// TIA Portal V18 export
DATA_BLOCK "DB_ALL_PROCESS_PARAMETERS"   // DB5000
{ S7_Optimized_Access := 'TRUE' }
// stored: AutoNumber false, MemoryReserve 1000
   VAR RETAIN
      "Choosen Recipe Number" : Bool;
      ACTUAL_CHOOSEN_TYPE : "UDT_OP10_Recipe_type";   // THERE IS ASCTUAL DATA READED OUT FROM LIBRARY OF 20 TYPES BELOW
      PRODUCT_TYPE : Array[1..10] of "UDT_OP10_Recipe_type";   // PACK OF TWENTY DIFFERENT TYPES PRODUCT AND THEIR PARAMETERS FOR THE PROCESS
   END_VAR
BEGIN
   ACTUAL_CHOOSEN_TYPE.Header.RecipeName := 'produkt 1';
   ACTUAL_CHOOSEN_TYPE.Header.RecipeID := 2;
   ACTUAL_CHOOSEN_TYPE.Header."Version" := 19629;
   ACTUAL_CHOOSEN_TYPE.Header.LastModified := DTL#2026-01-17-04:23:27.501;
   ACTUAL_CHOOSEN_TYPE.Header.PartType := 'additional  name';
   ACTUAL_CHOOSEN_TYPE.Process.Timers.Delay_glue_init_start := T#2S;
   ACTUAL_CHOOSEN_TYPE.Process.Timers.Delay_Medium := T#600MS;
   ACTUAL_CHOOSEN_TYPE.Process.Timers.Delay_Long := T#2S;
   ACTUAL_CHOOSEN_TYPE.Process.Timers.Cylinder_ActTime := T#6S;
   ACTUAL_CHOOSEN_TYPE.Process.Limits.RetryLimit := 3;
   ACTUAL_CHOOSEN_TYPE.Process.Press.B1_Program := 1;
   ACTUAL_CHOOSEN_TYPE.Process.Press.B2_Program := 1;
   ACTUAL_CHOOSEN_TYPE.Process.Vision.CGlueShaftIV3_Progs[1] := 16#0001;
   ACTUAL_CHOOSEN_TYPE.Process.Vision.CGlueShaftIV3_Progs[2] := 16#0002;
   ACTUAL_CHOOSEN_TYPE.Process.Vision.CGlueShaftIV3_Progs[3] := 16#0003;
   ACTUAL_CHOOSEN_TYPE.Process.Vision.CGlueShaftIV3_Progs[4] := 16#0004;
   ACTUAL_CHOOSEN_TYPE.Process.Vision.CGlueMagnetIV3_Prog := 16#0001;
   ACTUAL_CHOOSEN_TYPE.Process.Vision.CGlueProgram := 1;
   ACTUAL_CHOOSEN_TYPE."Tooling Code".A1_Table[1] := 'SZ23055-OP010-E-Compressor-ring1 Loading tooling-1';
   ACTUAL_CHOOSEN_TYPE."Tooling Code".A1_Table[2] := 'SZ23055-OP010-E-Compressor-ring1 Loading tooling-2';
   ACTUAL_CHOOSEN_TYPE."Tooling Code".A1_Table[3] := 'SZ23055-OP010-E-Compressor-ring1 Loading tooling-3';
   ACTUAL_CHOOSEN_TYPE."Tooling Code".A1_Table[4] := 'SZ23055-OP010-E-Compressor-ring1 Loading tooling-4';
   ACTUAL_CHOOSEN_TYPE."Tooling Code".A1_Table[5] := 'SZ23055-OP010-E-Compressor-ring1 Loading tooling-5';
   ACTUAL_CHOOSEN_TYPE."Tooling Code".A1_Table[6] := 'SZ23055-OP010-E-Compressor-ring1 Loading tooling-6';
   ACTUAL_CHOOSEN_TYPE."Tooling Code".A1_Table[7] := 'SZ23055-OP010-E-Compressor-ring1 Loading tooling-7';
   ACTUAL_CHOOSEN_TYPE."Tooling Code".A1_Table[8] := 'SZ23055-OP010-E-Compressor-ring1 Loading tooling-8';
   ACTUAL_CHOOSEN_TYPE."Tooling Code".A2_Table[1] := 'SZ23055-OP010-E-Compresspr-ring1 cutting tool';
   ACTUAL_CHOOSEN_TYPE."Tooling Code".A2_Table[2] := 'SZ23055-OP010-E-Compressor-Left NG tooling-1';
   ACTUAL_CHOOSEN_TYPE."Tooling Code".A2_Table[3] := 'SZ23055-OP010-E-Compressor-shaft Rotating scanning tooling-1';
   ACTUAL_CHOOSEN_TYPE."Tooling Code".A2_Table[4] := 'SZ23055-OP010-E-Compressor-ring1 Below Positioning fixture -1';
   ACTUAL_CHOOSEN_TYPE."Tooling Code".A2_Table[5] := 'SZ23055-OP010-E-Compressor-Point adhesive tooling-1';
   ACTUAL_CHOOSEN_TYPE."Tooling Code".A2_Table[6] := 'SZ23055-OP010-E-Compressor-ring1 Upper pressing fixture-1';
   ACTUAL_CHOOSEN_TYPE."Tooling Code".A2_Table[7] := 'SZ23055-OP010-E-Compresspr-ring2 cutting tool';
   ACTUAL_CHOOSEN_TYPE."Tooling Code".A2_Table[8] := 'SZ23055-OP010-E-Compressor-Right NG tooling-1';
   ACTUAL_CHOOSEN_TYPE."Tooling Code".ROB1_Shaft_Handling_Robot.Gripper."JAW TOOLING LEFT" := 'SZ23055-OP010-E-Compressor-robot1 ring1 Left clamping jaw tooling-1';
   ACTUAL_CHOOSEN_TYPE."Tooling Code".ROB1_Shaft_Handling_Robot.Gripper."JAW TOOLING RIGHT" := 'SZ23055-OP010-E-Compressor-robot1 ring1 Right clamping jaw tooling-2';
   ACTUAL_CHOOSEN_TYPE."Tooling Code".ROB1_Shaft_Handling_Robot.Gripper."SHAFT CLAMPING LEFT" := 'SZ23055-OP010-E-Compressor-robot1 shaft Left clamping jaw tooling-1';
   ACTUAL_CHOOSEN_TYPE."Tooling Code".ROB1_Shaft_Handling_Robot.Gripper."SHAFT CLAMPING RIGHT" := 'SZ23055-OP010-E-Compressor-robot1 shaft Right clamping jaw tooling-2';
   ACTUAL_CHOOSEN_TYPE."Tooling Code".ROB2_Main_Assembly_Robot.Gripper."JAW TOOLING LEFT" := 'SZ23055-OP010-E-Compressor-robot2 shaft Right clamping jaw tooling-2';
   ACTUAL_CHOOSEN_TYPE."Tooling Code".ROB2_Main_Assembly_Robot.Gripper."JAW TOOLING RIGHT" := 'SZ23055-OP010-E-Compressor-robot2 shaft Left clamping jaw tooling-1';
   ACTUAL_CHOOSEN_TYPE."Tooling Code".ROB2_Main_Assembly_Robot.Gripper."SHAFT CLAMPING LEFT" := 'SZ23055-OP010-E-Compressor-robot2 magnet Right clamping jaw tooling-2';
   ACTUAL_CHOOSEN_TYPE."Tooling Code".ROB2_Main_Assembly_Robot.Gripper."SHAFT CLAMPING RIGHT" := 'SZ23055-OP010-E-Compressor-robot2 magnet Right clamping jaw tooling-2';
   ACTUAL_CHOOSEN_TYPE."Tooling Code".ROB3_Unloading_Robot.Gripper."JAW TOOLING LEFT" := 'SZ23055-OP010-E-Compressor-robot3 ring2 Right clamping jaw tooling-2';
   ACTUAL_CHOOSEN_TYPE."Tooling Code".ROB3_Unloading_Robot.Gripper."JAW TOOLING RIGHT" := 'SZ23055-OP010-E-Compressor-robot3 ring2 Left clamping jaw tooling-1';
   ACTUAL_CHOOSEN_TYPE."Tooling Code".ROB3_Unloading_Robot.Gripper."SHAFT CLAMPING LEFT" := 'SZ23055-OP010-E-Compressor-robot3 shaft Left clamping jaw tooling-1';
   ACTUAL_CHOOSEN_TYPE."Tooling Code".ROB3_Unloading_Robot.Gripper."SHAFT CLAMPING RIGHT" := 'SZ23055-OP010-E-Compressor-robot3 shaft Right clamping jaw tooling-2';
   ACTUAL_CHOOSEN_TYPE."Tooling Code".A1_Fixtures.A1RingUnloadingFixtureCode := 'SZ23055-OP010-E-Compresspr-ring1 cutting tool';
   ACTUAL_CHOOSEN_TYPE."Tooling Code".A1_Fixtures.E1LoadingNGFixtureCode := 'SZ23055-OP010-E-Compressor-Left NG tooling-1';
   ACTUAL_CHOOSEN_TYPE."Tooling Code".A1_Fixtures.ShaftScanFixtureCode := 'SZ23055-OP010-E-Compressor-shaft Rotating scanning tooling-1';
   ACTUAL_CHOOSEN_TYPE."Tooling Code".A1_Fixtures.B1PressFixtureCode := 'SZ23055-OP010-E-Compressor-ring1 Below Positioning fixture -1';
   ACTUAL_CHOOSEN_TYPE."Tooling Code".A1_Fixtures.CGlueFixtureCode := 'SZ23055-OP010-E-Compressor-Point adhesive tooling-1';
   ACTUAL_CHOOSEN_TYPE."Tooling Code".A1_Fixtures.B1PressCylFixtureCode := 'SZ23055-OP010-E-Compressor-ring1 Upper pressing fixture-1';
   ACTUAL_CHOOSEN_TYPE."Tooling Code".A2_Fixtures.A2RingUnloadingFixtureCode := 'SZ23055-OP010-E-Compresspr-ring2 cutting tool';
   ACTUAL_CHOOSEN_TYPE."Tooling Code".A2_Fixtures.E2UnloadingNGFixtureCode := 'SZ23055-OP010-E-Compressor-Right NG tooling-1';
   ACTUAL_CHOOSEN_TYPE."Tooling Code".A2_Fixtures.B2PressFixtureCode := 'SZ23055-OP010-E-Compressor-ring2 Below Positioning fixture -1';
   ACTUAL_CHOOSEN_TYPE."Tooling Code".A2_Fixtures.CGlueNGFixtureCode := 'SZ23055-OP010-E-Compressor-NG middle shift tooling-1';
   ACTUAL_CHOOSEN_TYPE."Tooling Code".A2_Fixtures.B2PressCylFixtureCode := 'SZ23055-OP010-E-Compressor-ring2 Upper pressing fixture-1';
   ACTUAL_CHOOSEN_TYPE.Motion.Gluing_Nozzle_Z.Position[1].Pos := 143.76;
   ACTUAL_CHOOSEN_TYPE.Motion.Gluing_Nozzle_Z.Position[2].Pos := 139.11;
   ACTUAL_CHOOSEN_TYPE.Motion.Gluing_Nozzle_Z.Position[3].Pos := 131.98;
   ACTUAL_CHOOSEN_TYPE.Motion.Gluing_Nozzle_Z.Position[4].Pos := 127.89;
   ACTUAL_CHOOSEN_TYPE.Motion.Gluing_Nozzle_Z.Position[6].Pos := 127.0;
   ACTUAL_CHOOSEN_TYPE.Motion.Gluing_Nozzle_Z.Position[7].Pos := 48.11;
   ACTUAL_CHOOSEN_TYPE.Motion.Gluing_Nozzle_Z.Position[9].Pos := 123.0;
   ACTUAL_CHOOSEN_TYPE.Motion.Gluing_Nozzle_Z.Position[1..4].Vel := 200;
   ACTUAL_CHOOSEN_TYPE.Motion.Gluing_Nozzle_Z.Position[6..9].Vel := 200;
   ACTUAL_CHOOSEN_TYPE.Motion.Gluing_Nozzle_X.Position[1].Pos := 2.34;
   ACTUAL_CHOOSEN_TYPE.Motion.Gluing_Nozzle_X.Position[2].Pos := 76.0;
   ACTUAL_CHOOSEN_TYPE.Motion.Gluing_Nozzle_X.Position[3..6].Pos := 84.69;
   ACTUAL_CHOOSEN_TYPE.Motion.Gluing_Nozzle_X.Position[7].Pos := 85.0;
   ACTUAL_CHOOSEN_TYPE.Motion.Gluing_Nozzle_X.Position[8].Pos := 88.53;
   ACTUAL_CHOOSEN_TYPE.Motion.Gluing_Nozzle_X.Position[1..8].Vel := 200;
   ACTUAL_CHOOSEN_TYPE.Motion.Gluing_Nozzle_Y.Position[1..5].Pos := 115.47;
   ACTUAL_CHOOSEN_TYPE.Motion.Gluing_Nozzle_Y.Position[6].Pos := 110.18;
   ACTUAL_CHOOSEN_TYPE.Motion.Gluing_Nozzle_Y.Position[7].Pos := 60.52;
   ACTUAL_CHOOSEN_TYPE.Motion.Gluing_Nozzle_Y.Position[8].Pos := 80.0;
   ACTUAL_CHOOSEN_TYPE.Motion.Gluing_Nozzle_Y.Position[1..7].Vel := 200;
   ACTUAL_CHOOSEN_TYPE.Motion.Gluing_Nozzle_Y.Position[8].Vel := 100;
   ACTUAL_CHOOSEN_TYPE.Motion.Ring_Turntable_Axis_1.Position[1].Pos := 3419;
   ACTUAL_CHOOSEN_TYPE.Motion.Ring_Turntable_Axis_1.Position[2].Pos := 48386;
   ACTUAL_CHOOSEN_TYPE.Motion.Ring_Turntable_Axis_1.Position[3].Pos := 93294;
   ACTUAL_CHOOSEN_TYPE.Motion.Ring_Turntable_Axis_1.Position[4].Pos := 138335;
   ACTUAL_CHOOSEN_TYPE.Motion.Ring_Turntable_Axis_1.Position[5].Pos := 183464;
   ACTUAL_CHOOSEN_TYPE.Motion.Ring_Turntable_Axis_1.Position[6].Pos := 228443;
   ACTUAL_CHOOSEN_TYPE.Motion.Ring_Turntable_Axis_1.Position[7].Pos := 273535;
   ACTUAL_CHOOSEN_TYPE.Motion.Ring_Turntable_Axis_1.Position[8].Pos := 318250;
   ACTUAL_CHOOSEN_TYPE.Motion.Ring_Turntable_Axis_1.Position[1..8].Vel := 10000;
   ACTUAL_CHOOSEN_TYPE.Motion.Shaft_Scan_Turntable_Axis.Position[2].Pos := 450000;
   ACTUAL_CHOOSEN_TYPE.Motion.Shaft_Scan_Turntable_Axis.Position[3].Pos := 900000;
   ACTUAL_CHOOSEN_TYPE.Motion.Shaft_Scan_Turntable_Axis.Position[4].Pos := 135000;
   ACTUAL_CHOOSEN_TYPE.Motion.Shaft_Scan_Turntable_Axis.Position[5].Pos := 180000;
   ACTUAL_CHOOSEN_TYPE.Motion.Shaft_Scan_Turntable_Axis.Position[6].Pos := 225000;
   ACTUAL_CHOOSEN_TYPE.Motion.Shaft_Scan_Turntable_Axis.Position[7].Pos := 270000;
   ACTUAL_CHOOSEN_TYPE.Motion.Shaft_Scan_Turntable_Axis.Position[8].Pos := 315000;
   ACTUAL_CHOOSEN_TYPE.Motion.Shaft_Scan_Turntable_Axis.Position[1..8].Vel := 10000;
   ACTUAL_CHOOSEN_TYPE.Motion.Gluing_Rotary_Jig_Axis.Position[3..6].Pos := 680000;
   ACTUAL_CHOOSEN_TYPE.Motion.Gluing_Rotary_Jig_Axis.Position[7].Pos := 90000;
   ACTUAL_CHOOSEN_TYPE.Motion.Gluing_Rotary_Jig_Axis.Position[8].Pos := 180000;
   ACTUAL_CHOOSEN_TYPE.Motion.Gluing_Rotary_Jig_Axis.Position[9].Pos := 270000;
   ACTUAL_CHOOSEN_TYPE.Motion.Gluing_Rotary_Jig_Axis.Position[1..2].Vel := 20000;
   ACTUAL_CHOOSEN_TYPE.Motion.Gluing_Rotary_Jig_Axis.Position[3..9].Vel := 10000;
   ACTUAL_CHOOSEN_TYPE.Motion.Ring_Turntable_Axis_2.Position[1].Pos := 3585;
   ACTUAL_CHOOSEN_TYPE.Motion.Ring_Turntable_Axis_2.Position[2].Pos := 48610;
   ACTUAL_CHOOSEN_TYPE.Motion.Ring_Turntable_Axis_2.Position[3].Pos := 93637;
   ACTUAL_CHOOSEN_TYPE.Motion.Ring_Turntable_Axis_2.Position[4].Pos := 138606;
   ACTUAL_CHOOSEN_TYPE.Motion.Ring_Turntable_Axis_2.Position[5].Pos := 183388;
   ACTUAL_CHOOSEN_TYPE.Motion.Ring_Turntable_Axis_2.Position[6].Pos := 228458;
   ACTUAL_CHOOSEN_TYPE.Motion.Ring_Turntable_Axis_2.Position[7].Pos := 273513;
   ACTUAL_CHOOSEN_TYPE.Motion.Ring_Turntable_Axis_2.Position[8].Pos := 318501;
   ACTUAL_CHOOSEN_TYPE.Motion.Ring_Turntable_Axis_2.Position[1..8].Vel := 10000;
   PRODUCT_TYPE[1].Header.RecipeName := 'produkt 1';
   PRODUCT_TYPE[3].Header.RecipeName := 'produkt 1';
   PRODUCT_TYPE[10].Header.RecipeName := 'produkt 1';
   PRODUCT_TYPE[1].Header.RecipeID := 1;
   PRODUCT_TYPE[3].Header.RecipeID := 1;
   PRODUCT_TYPE[10].Header.RecipeID := 1;
   PRODUCT_TYPE[1].Header."Version" := 1;
   PRODUCT_TYPE[3].Header."Version" := 1;
   PRODUCT_TYPE[10].Header."Version" := 1;
   PRODUCT_TYPE[1].Header.LastModified := DTL#2026-01-17-04:23:27.501;
   PRODUCT_TYPE[3].Header.LastModified := DTL#2026-01-17-04:23:27.501;
   PRODUCT_TYPE[10].Header.LastModified := DTL#2026-01-17-04:23:27.501;
   PRODUCT_TYPE[1].Header.PartType := 'additional  name';
   PRODUCT_TYPE[3].Header.PartType := 'additional  name';
   PRODUCT_TYPE[10].Header.PartType := 'additional  name';
   PRODUCT_TYPE[1].Process.Timers.Delay_glue_init_start := T#2S;
   PRODUCT_TYPE[2].Process.Timers.Delay_glue_init_start := T#0MS;
   PRODUCT_TYPE[3].Process.Timers.Delay_glue_init_start := T#300MS;
   PRODUCT_TYPE[4..9].Process.Timers.Delay_glue_init_start := T#0MS;
   PRODUCT_TYPE[10].Process.Timers.Delay_glue_init_start := T#2S;
   PRODUCT_TYPE[1].Process.Timers.Delay_Medium := T#600MS;
   PRODUCT_TYPE[3].Process.Timers.Delay_Medium := T#600MS;
   PRODUCT_TYPE[10].Process.Timers.Delay_Medium := T#600MS;
   PRODUCT_TYPE[1].Process.Timers.Delay_Long := T#2S;
   PRODUCT_TYPE[3].Process.Timers.Delay_Long := T#2S;
   PRODUCT_TYPE[10].Process.Timers.Delay_Long := T#2S;
   PRODUCT_TYPE[1].Process.Timers.Cylinder_ActTime := T#6S;
   PRODUCT_TYPE[3].Process.Timers.Cylinder_ActTime := T#6S;
   PRODUCT_TYPE[10].Process.Timers.Cylinder_ActTime := T#6S;
   PRODUCT_TYPE[1].Process.Limits.RetryLimit := 3;
   PRODUCT_TYPE[3].Process.Limits.RetryLimit := 3;
   PRODUCT_TYPE[10].Process.Limits.RetryLimit := 3;
   PRODUCT_TYPE[1].Process.Press.B1_Program := 1;
   PRODUCT_TYPE[3].Process.Press.B1_Program := 1;
   PRODUCT_TYPE[10].Process.Press.B1_Program := 1;
   PRODUCT_TYPE[1].Process.Press.B2_Program := 1;
   PRODUCT_TYPE[3].Process.Press.B2_Program := 1;
   PRODUCT_TYPE[10].Process.Press.B2_Program := 1;
   PRODUCT_TYPE[1].Process.Vision.CGlueShaftIV3_Progs[1] := 16#0001;
   PRODUCT_TYPE[1].Process.Vision.CGlueShaftIV3_Progs[2] := 16#0002;
   PRODUCT_TYPE[1].Process.Vision.CGlueShaftIV3_Progs[3] := 16#0003;
   PRODUCT_TYPE[1].Process.Vision.CGlueShaftIV3_Progs[4] := 16#0004;
   PRODUCT_TYPE[3].Process.Vision.CGlueShaftIV3_Progs[1] := 16#0001;
   PRODUCT_TYPE[3].Process.Vision.CGlueShaftIV3_Progs[2] := 16#0002;
   PRODUCT_TYPE[3].Process.Vision.CGlueShaftIV3_Progs[3] := 16#0003;
   PRODUCT_TYPE[3].Process.Vision.CGlueShaftIV3_Progs[4] := 16#0004;
   PRODUCT_TYPE[10].Process.Vision.CGlueShaftIV3_Progs[1] := 16#0001;
   PRODUCT_TYPE[10].Process.Vision.CGlueShaftIV3_Progs[2] := 16#0002;
   PRODUCT_TYPE[10].Process.Vision.CGlueShaftIV3_Progs[3] := 16#0003;
   PRODUCT_TYPE[10].Process.Vision.CGlueShaftIV3_Progs[4] := 16#0004;
   PRODUCT_TYPE[1].Process.Vision.CGlueMagnetIV3_Prog := 16#0001;
   PRODUCT_TYPE[3].Process.Vision.CGlueMagnetIV3_Prog := 16#0001;
   PRODUCT_TYPE[10].Process.Vision.CGlueMagnetIV3_Prog := 16#0001;
   PRODUCT_TYPE[1].Process.Vision.CGlueProgram := 1;
   PRODUCT_TYPE[3].Process.Vision.CGlueProgram := 1;
   PRODUCT_TYPE[10].Process.Vision.CGlueProgram := 1;
   PRODUCT_TYPE[1]."Tooling Code".A1_Table[1] := 'SZ23055-OP010-E-Compressor-ring1 Loading tooling-1';
   PRODUCT_TYPE[1]."Tooling Code".A1_Table[2] := 'SZ23055-OP010-E-Compressor-ring1 Loading tooling-2';
   PRODUCT_TYPE[1]."Tooling Code".A1_Table[3] := 'SZ23055-OP010-E-Compressor-ring1 Loading tooling-3';
   PRODUCT_TYPE[1]."Tooling Code".A1_Table[4] := 'SZ23055-OP010-E-Compressor-ring1 Loading tooling-4';
   PRODUCT_TYPE[1]."Tooling Code".A1_Table[5] := 'SZ23055-OP010-E-Compressor-ring1 Loading tooling-5';
   PRODUCT_TYPE[1]."Tooling Code".A1_Table[6] := 'SZ23055-OP010-E-Compressor-ring1 Loading tooling-6';
   PRODUCT_TYPE[1]."Tooling Code".A1_Table[7] := 'SZ23055-OP010-E-Compressor-ring1 Loading tooling-7';
   PRODUCT_TYPE[1]."Tooling Code".A1_Table[8] := 'SZ23055-OP010-E-Compressor-ring1 Loading tooling-8';
   PRODUCT_TYPE[3]."Tooling Code".A1_Table[1] := 'SZ23055-OP010-E-Compressor-ring1 Loading tooling-1';
   PRODUCT_TYPE[3]."Tooling Code".A1_Table[2] := 'SZ23055-OP010-E-Compressor-ring1 Loading tooling-2';
   PRODUCT_TYPE[3]."Tooling Code".A1_Table[3] := 'SZ23055-OP010-E-Compressor-ring1 Loading tooling-3';
   PRODUCT_TYPE[3]."Tooling Code".A1_Table[4] := 'SZ23055-OP010-E-Compressor-ring1 Loading tooling-4';
   PRODUCT_TYPE[3]."Tooling Code".A1_Table[5] := 'SZ23055-OP010-E-Compressor-ring1 Loading tooling-5';
   PRODUCT_TYPE[3]."Tooling Code".A1_Table[6] := 'SZ23055-OP010-E-Compressor-ring1 Loading tooling-6';
   PRODUCT_TYPE[3]."Tooling Code".A1_Table[7] := 'SZ23055-OP010-E-Compressor-ring1 Loading tooling-7';
   PRODUCT_TYPE[3]."Tooling Code".A1_Table[8] := 'SZ23055-OP010-E-Compressor-ring1 Loading tooling-8';
   PRODUCT_TYPE[10]."Tooling Code".A1_Table[1] := 'SZ23055-OP010-E-Compressor-ring1 Loading tooling-1';
   PRODUCT_TYPE[10]."Tooling Code".A1_Table[2] := 'SZ23055-OP010-E-Compressor-ring1 Loading tooling-2';
   PRODUCT_TYPE[10]."Tooling Code".A1_Table[3] := 'SZ23055-OP010-E-Compressor-ring1 Loading tooling-3';
   PRODUCT_TYPE[10]."Tooling Code".A1_Table[4] := 'SZ23055-OP010-E-Compressor-ring1 Loading tooling-4';
   PRODUCT_TYPE[10]."Tooling Code".A1_Table[5] := 'SZ23055-OP010-E-Compressor-ring1 Loading tooling-5';
   PRODUCT_TYPE[10]."Tooling Code".A1_Table[6] := 'SZ23055-OP010-E-Compressor-ring1 Loading tooling-6';
   PRODUCT_TYPE[10]."Tooling Code".A1_Table[7] := 'SZ23055-OP010-E-Compressor-ring1 Loading tooling-7';
   PRODUCT_TYPE[10]."Tooling Code".A1_Table[8] := 'SZ23055-OP010-E-Compressor-ring1 Loading tooling-8';
   PRODUCT_TYPE[1]."Tooling Code".A2_Table[1] := 'SZ23055-OP010-E-Compresspr-ring1 cutting tool';
   PRODUCT_TYPE[1]."Tooling Code".A2_Table[2] := 'SZ23055-OP010-E-Compressor-Left NG tooling-1';
   PRODUCT_TYPE[1]."Tooling Code".A2_Table[3] := 'SZ23055-OP010-E-Compressor-shaft Rotating scanning tooling-1';
   PRODUCT_TYPE[1]."Tooling Code".A2_Table[4] := 'SZ23055-OP010-E-Compressor-ring1 Below Positioning fixture -1';
   PRODUCT_TYPE[1]."Tooling Code".A2_Table[5] := 'SZ23055-OP010-E-Compressor-Point adhesive tooling-1';
   PRODUCT_TYPE[1]."Tooling Code".A2_Table[6] := 'SZ23055-OP010-E-Compressor-ring1 Upper pressing fixture-1';
   PRODUCT_TYPE[1]."Tooling Code".A2_Table[7] := 'SZ23055-OP010-E-Compresspr-ring2 cutting tool';
   PRODUCT_TYPE[1]."Tooling Code".A2_Table[8] := 'SZ23055-OP010-E-Compressor-Right NG tooling-1';
   PRODUCT_TYPE[3]."Tooling Code".A2_Table[1] := 'SZ23055-OP010-E-Compresspr-ring1 cutting tool';
   PRODUCT_TYPE[3]."Tooling Code".A2_Table[2] := 'SZ23055-OP010-E-Compressor-Left NG tooling-1';
   PRODUCT_TYPE[3]."Tooling Code".A2_Table[3] := 'SZ23055-OP010-E-Compressor-shaft Rotating scanning tooling-1';
   PRODUCT_TYPE[3]."Tooling Code".A2_Table[4] := 'SZ23055-OP010-E-Compressor-ring1 Below Positioning fixture -1';
   PRODUCT_TYPE[3]."Tooling Code".A2_Table[5] := 'SZ23055-OP010-E-Compressor-Point adhesive tooling-1';
   PRODUCT_TYPE[3]."Tooling Code".A2_Table[6] := 'SZ23055-OP010-E-Compressor-ring1 Upper pressing fixture-1';
   PRODUCT_TYPE[3]."Tooling Code".A2_Table[7] := 'SZ23055-OP010-E-Compresspr-ring2 cutting tool';
   PRODUCT_TYPE[3]."Tooling Code".A2_Table[8] := 'SZ23055-OP010-E-Compressor-Right NG tooling-1';
   PRODUCT_TYPE[10]."Tooling Code".A2_Table[1] := 'SZ23055-OP010-E-Compresspr-ring1 cutting tool';
   PRODUCT_TYPE[10]."Tooling Code".A2_Table[2] := 'SZ23055-OP010-E-Compressor-Left NG tooling-1';
   PRODUCT_TYPE[10]."Tooling Code".A2_Table[3] := 'SZ23055-OP010-E-Compressor-shaft Rotating scanning tooling-1';
   PRODUCT_TYPE[10]."Tooling Code".A2_Table[4] := 'SZ23055-OP010-E-Compressor-ring1 Below Positioning fixture -1';
   PRODUCT_TYPE[10]."Tooling Code".A2_Table[5] := 'SZ23055-OP010-E-Compressor-Point adhesive tooling-1';
   PRODUCT_TYPE[10]."Tooling Code".A2_Table[6] := 'SZ23055-OP010-E-Compressor-ring1 Upper pressing fixture-1';
   PRODUCT_TYPE[10]."Tooling Code".A2_Table[7] := 'SZ23055-OP010-E-Compresspr-ring2 cutting tool';
   PRODUCT_TYPE[10]."Tooling Code".A2_Table[8] := 'SZ23055-OP010-E-Compressor-Right NG tooling-1';
   PRODUCT_TYPE[1]."Tooling Code".ROB1_Shaft_Handling_Robot.Gripper."JAW TOOLING LEFT" := 'SZ23055-OP010-E-Compressor-robot1 ring1 Left clamping jaw tooling-1';
   PRODUCT_TYPE[3]."Tooling Code".ROB1_Shaft_Handling_Robot.Gripper."JAW TOOLING LEFT" := 'SZ23055-OP010-E-Compressor-robot1 ring1 Left clamping jaw tooling-1';
   PRODUCT_TYPE[10]."Tooling Code".ROB1_Shaft_Handling_Robot.Gripper."JAW TOOLING LEFT" := 'SZ23055-OP010-E-Compressor-robot1 ring1 Left clamping jaw tooling-1';
   PRODUCT_TYPE[1]."Tooling Code".ROB1_Shaft_Handling_Robot.Gripper."JAW TOOLING RIGHT" := 'SZ23055-OP010-E-Compressor-robot1 ring1 Right clamping jaw tooling-2';
   PRODUCT_TYPE[3]."Tooling Code".ROB1_Shaft_Handling_Robot.Gripper."JAW TOOLING RIGHT" := 'SZ23055-OP010-E-Compressor-robot1 ring1 Right clamping jaw tooling-2';
   PRODUCT_TYPE[10]."Tooling Code".ROB1_Shaft_Handling_Robot.Gripper."JAW TOOLING RIGHT" := 'SZ23055-OP010-E-Compressor-robot1 ring1 Right clamping jaw tooling-2';
   PRODUCT_TYPE[1]."Tooling Code".ROB1_Shaft_Handling_Robot.Gripper."SHAFT CLAMPING LEFT" := 'SZ23055-OP010-E-Compressor-robot1 shaft Left clamping jaw tooling-1';
   PRODUCT_TYPE[3]."Tooling Code".ROB1_Shaft_Handling_Robot.Gripper."SHAFT CLAMPING LEFT" := 'SZ23055-OP010-E-Compressor-robot1 shaft Left clamping jaw tooling-1';
   PRODUCT_TYPE[10]."Tooling Code".ROB1_Shaft_Handling_Robot.Gripper."SHAFT CLAMPING LEFT" := 'SZ23055-OP010-E-Compressor-robot1 shaft Left clamping jaw tooling-1';
   PRODUCT_TYPE[1]."Tooling Code".ROB1_Shaft_Handling_Robot.Gripper."SHAFT CLAMPING RIGHT" := 'SZ23055-OP010-E-Compressor-robot1 shaft Right clamping jaw tooling-2';
   PRODUCT_TYPE[3]."Tooling Code".ROB1_Shaft_Handling_Robot.Gripper."SHAFT CLAMPING RIGHT" := 'SZ23055-OP010-E-Compressor-robot1 shaft Right clamping jaw tooling-2';
   PRODUCT_TYPE[10]."Tooling Code".ROB1_Shaft_Handling_Robot.Gripper."SHAFT CLAMPING RIGHT" := 'SZ23055-OP010-E-Compressor-robot1 shaft Right clamping jaw tooling-2';
   PRODUCT_TYPE[1]."Tooling Code".ROB2_Main_Assembly_Robot.Gripper."JAW TOOLING LEFT" := 'SZ23055-OP010-E-Compressor-robot2 shaft Right clamping jaw tooling-2';
   PRODUCT_TYPE[3]."Tooling Code".ROB2_Main_Assembly_Robot.Gripper."JAW TOOLING LEFT" := 'SZ23055-OP010-E-Compressor-robot2 shaft Right clamping jaw tooling-2';
   PRODUCT_TYPE[10]."Tooling Code".ROB2_Main_Assembly_Robot.Gripper."JAW TOOLING LEFT" := 'SZ23055-OP010-E-Compressor-robot2 shaft Right clamping jaw tooling-2';
   PRODUCT_TYPE[1]."Tooling Code".ROB2_Main_Assembly_Robot.Gripper."JAW TOOLING RIGHT" := 'SZ23055-OP010-E-Compressor-robot2 shaft Left clamping jaw tooling-1';
   PRODUCT_TYPE[3]."Tooling Code".ROB2_Main_Assembly_Robot.Gripper."JAW TOOLING RIGHT" := 'SZ23055-OP010-E-Compressor-robot2 shaft Left clamping jaw tooling-1';
   PRODUCT_TYPE[10]."Tooling Code".ROB2_Main_Assembly_Robot.Gripper."JAW TOOLING RIGHT" := 'SZ23055-OP010-E-Compressor-robot2 shaft Left clamping jaw tooling-1';
   PRODUCT_TYPE[1]."Tooling Code".ROB2_Main_Assembly_Robot.Gripper."SHAFT CLAMPING LEFT" := 'SZ23055-OP010-E-Compressor-robot2 magnet Right clamping jaw tooling-2';
   PRODUCT_TYPE[3]."Tooling Code".ROB2_Main_Assembly_Robot.Gripper."SHAFT CLAMPING LEFT" := 'SZ23055-OP010-E-Compressor-robot2 magnet Right clamping jaw tooling-2';
   PRODUCT_TYPE[10]."Tooling Code".ROB2_Main_Assembly_Robot.Gripper."SHAFT CLAMPING LEFT" := 'SZ23055-OP010-E-Compressor-robot2 magnet Right clamping jaw tooling-2';
   PRODUCT_TYPE[1]."Tooling Code".ROB2_Main_Assembly_Robot.Gripper."SHAFT CLAMPING RIGHT" := 'SZ23055-OP010-E-Compressor-robot2 magnet Right clamping jaw tooling-2';
   PRODUCT_TYPE[3]."Tooling Code".ROB2_Main_Assembly_Robot.Gripper."SHAFT CLAMPING RIGHT" := 'SZ23055-OP010-E-Compressor-robot2 magnet Right clamping jaw tooling-2';
   PRODUCT_TYPE[10]."Tooling Code".ROB2_Main_Assembly_Robot.Gripper."SHAFT CLAMPING RIGHT" := 'SZ23055-OP010-E-Compressor-robot2 magnet Right clamping jaw tooling-2';
   PRODUCT_TYPE[1]."Tooling Code".ROB3_Unloading_Robot.Gripper."JAW TOOLING LEFT" := 'SZ23055-OP010-E-Compressor-robot3 ring2 Right clamping jaw tooling-2';
   PRODUCT_TYPE[3]."Tooling Code".ROB3_Unloading_Robot.Gripper."JAW TOOLING LEFT" := 'SZ23055-OP010-E-Compressor-robot3 ring2 Right clamping jaw tooling-2';
   PRODUCT_TYPE[10]."Tooling Code".ROB3_Unloading_Robot.Gripper."JAW TOOLING LEFT" := 'SZ23055-OP010-E-Compressor-robot3 ring2 Right clamping jaw tooling-2';
   PRODUCT_TYPE[1]."Tooling Code".ROB3_Unloading_Robot.Gripper."JAW TOOLING RIGHT" := 'SZ23055-OP010-E-Compressor-robot3 ring2 Left clamping jaw tooling-1';
   PRODUCT_TYPE[3]."Tooling Code".ROB3_Unloading_Robot.Gripper."JAW TOOLING RIGHT" := 'SZ23055-OP010-E-Compressor-robot3 ring2 Left clamping jaw tooling-1';
   PRODUCT_TYPE[10]."Tooling Code".ROB3_Unloading_Robot.Gripper."JAW TOOLING RIGHT" := 'SZ23055-OP010-E-Compressor-robot3 ring2 Left clamping jaw tooling-1';
   PRODUCT_TYPE[1]."Tooling Code".ROB3_Unloading_Robot.Gripper."SHAFT CLAMPING LEFT" := 'SZ23055-OP010-E-Compressor-robot3 shaft Left clamping jaw tooling-1';
   PRODUCT_TYPE[3]."Tooling Code".ROB3_Unloading_Robot.Gripper."SHAFT CLAMPING LEFT" := 'SZ23055-OP010-E-Compressor-robot3 shaft Left clamping jaw tooling-1';
   PRODUCT_TYPE[10]."Tooling Code".ROB3_Unloading_Robot.Gripper."SHAFT CLAMPING LEFT" := 'SZ23055-OP010-E-Compressor-robot3 shaft Left clamping jaw tooling-1';
   PRODUCT_TYPE[1]."Tooling Code".ROB3_Unloading_Robot.Gripper."SHAFT CLAMPING RIGHT" := 'SZ23055-OP010-E-Compressor-robot3 shaft Right clamping jaw tooling-2';
   PRODUCT_TYPE[3]."Tooling Code".ROB3_Unloading_Robot.Gripper."SHAFT CLAMPING RIGHT" := 'SZ23055-OP010-E-Compressor-robot3 shaft Right clamping jaw tooling-2';
   PRODUCT_TYPE[10]."Tooling Code".ROB3_Unloading_Robot.Gripper."SHAFT CLAMPING RIGHT" := 'SZ23055-OP010-E-Compressor-robot3 shaft Right clamping jaw tooling-2';
   PRODUCT_TYPE[1]."Tooling Code".A1_Fixtures.A1RingUnloadingFixtureCode := 'SZ23055-OP010-E-Compresspr-ring1 cutting tool';
   PRODUCT_TYPE[3]."Tooling Code".A1_Fixtures.A1RingUnloadingFixtureCode := 'SZ23055-OP010-E-Compresspr-ring1 cutting tool';
   PRODUCT_TYPE[10]."Tooling Code".A1_Fixtures.A1RingUnloadingFixtureCode := 'SZ23055-OP010-E-Compresspr-ring1 cutting tool';
   PRODUCT_TYPE[1]."Tooling Code".A1_Fixtures.E1LoadingNGFixtureCode := 'SZ23055-OP010-E-Compressor-Left NG tooling-1';
   PRODUCT_TYPE[3]."Tooling Code".A1_Fixtures.E1LoadingNGFixtureCode := 'SZ23055-OP010-E-Compressor-Left NG tooling-1';
   PRODUCT_TYPE[10]."Tooling Code".A1_Fixtures.E1LoadingNGFixtureCode := 'SZ23055-OP010-E-Compressor-Left NG tooling-1';
   PRODUCT_TYPE[1]."Tooling Code".A1_Fixtures.ShaftScanFixtureCode := 'SZ23055-OP010-E-Compressor-shaft Rotating scanning tooling-1';
   PRODUCT_TYPE[3]."Tooling Code".A1_Fixtures.ShaftScanFixtureCode := 'SZ23055-OP010-E-Compressor-shaft Rotating scanning tooling-1';
   PRODUCT_TYPE[10]."Tooling Code".A1_Fixtures.ShaftScanFixtureCode := 'SZ23055-OP010-E-Compressor-shaft Rotating scanning tooling-1';
   PRODUCT_TYPE[1]."Tooling Code".A1_Fixtures.B1PressFixtureCode := 'SZ23055-OP010-E-Compressor-ring1 Below Positioning fixture -1';
   PRODUCT_TYPE[3]."Tooling Code".A1_Fixtures.B1PressFixtureCode := 'SZ23055-OP010-E-Compressor-ring1 Below Positioning fixture -1';
   PRODUCT_TYPE[10]."Tooling Code".A1_Fixtures.B1PressFixtureCode := 'SZ23055-OP010-E-Compressor-ring1 Below Positioning fixture -1';
   PRODUCT_TYPE[1]."Tooling Code".A1_Fixtures.CGlueFixtureCode := 'SZ23055-OP010-E-Compressor-Point adhesive tooling-1';
   PRODUCT_TYPE[3]."Tooling Code".A1_Fixtures.CGlueFixtureCode := 'SZ23055-OP010-E-Compressor-Point adhesive tooling-1';
   PRODUCT_TYPE[10]."Tooling Code".A1_Fixtures.CGlueFixtureCode := 'SZ23055-OP010-E-Compressor-Point adhesive tooling-1';
   PRODUCT_TYPE[1]."Tooling Code".A1_Fixtures.B1PressCylFixtureCode := 'SZ23055-OP010-E-Compressor-ring1 Upper pressing fixture-1';
   PRODUCT_TYPE[3]."Tooling Code".A1_Fixtures.B1PressCylFixtureCode := 'SZ23055-OP010-E-Compressor-ring1 Upper pressing fixture-1';
   PRODUCT_TYPE[10]."Tooling Code".A1_Fixtures.B1PressCylFixtureCode := 'SZ23055-OP010-E-Compressor-ring1 Upper pressing fixture-1';
   PRODUCT_TYPE[1]."Tooling Code".A2_Fixtures.A2RingUnloadingFixtureCode := 'SZ23055-OP010-E-Compresspr-ring2 cutting tool';
   PRODUCT_TYPE[3]."Tooling Code".A2_Fixtures.A2RingUnloadingFixtureCode := 'SZ23055-OP010-E-Compresspr-ring2 cutting tool';
   PRODUCT_TYPE[10]."Tooling Code".A2_Fixtures.A2RingUnloadingFixtureCode := 'SZ23055-OP010-E-Compresspr-ring2 cutting tool';
   PRODUCT_TYPE[1]."Tooling Code".A2_Fixtures.E2UnloadingNGFixtureCode := 'SZ23055-OP010-E-Compressor-Right NG tooling-1';
   PRODUCT_TYPE[3]."Tooling Code".A2_Fixtures.E2UnloadingNGFixtureCode := 'SZ23055-OP010-E-Compressor-Right NG tooling-1';
   PRODUCT_TYPE[10]."Tooling Code".A2_Fixtures.E2UnloadingNGFixtureCode := 'SZ23055-OP010-E-Compressor-Right NG tooling-1';
   PRODUCT_TYPE[1]."Tooling Code".A2_Fixtures.B2PressFixtureCode := 'SZ23055-OP010-E-Compressor-ring2 Below Positioning fixture -1';
   PRODUCT_TYPE[3]."Tooling Code".A2_Fixtures.B2PressFixtureCode := 'SZ23055-OP010-E-Compressor-ring2 Below Positioning fixture -1';
   PRODUCT_TYPE[10]."Tooling Code".A2_Fixtures.B2PressFixtureCode := 'SZ23055-OP010-E-Compressor-ring2 Below Positioning fixture -1';
   PRODUCT_TYPE[1]."Tooling Code".A2_Fixtures.CGlueNGFixtureCode := 'SZ23055-OP010-E-Compressor-NG middle shift tooling-1';
   PRODUCT_TYPE[3]."Tooling Code".A2_Fixtures.CGlueNGFixtureCode := 'SZ23055-OP010-E-Compressor-NG middle shift tooling-1';
   PRODUCT_TYPE[10]."Tooling Code".A2_Fixtures.CGlueNGFixtureCode := 'SZ23055-OP010-E-Compressor-NG middle shift tooling-1';
   PRODUCT_TYPE[1]."Tooling Code".A2_Fixtures.B2PressCylFixtureCode := 'SZ23055-OP010-E-Compressor-ring2 Upper pressing fixture-1';
   PRODUCT_TYPE[3]."Tooling Code".A2_Fixtures.B2PressCylFixtureCode := 'SZ23055-OP010-E-Compressor-ring2 Upper pressing fixture-1';
   PRODUCT_TYPE[10]."Tooling Code".A2_Fixtures.B2PressCylFixtureCode := 'SZ23055-OP010-E-Compressor-ring2 Upper pressing fixture-1';
   PRODUCT_TYPE[1].Motion.Gluing_Nozzle_Z.Position[1].Pos := 143.76;
   PRODUCT_TYPE[1].Motion.Gluing_Nozzle_Z.Position[2].Pos := 139.11;
   PRODUCT_TYPE[1].Motion.Gluing_Nozzle_Z.Position[3].Pos := 131.98;
   PRODUCT_TYPE[1].Motion.Gluing_Nozzle_Z.Position[4].Pos := 127.89;
   PRODUCT_TYPE[1].Motion.Gluing_Nozzle_Z.Position[6].Pos := 127.0;
   PRODUCT_TYPE[1].Motion.Gluing_Nozzle_Z.Position[7].Pos := 48.11;
   PRODUCT_TYPE[1].Motion.Gluing_Nozzle_Z.Position[9].Pos := 123.0;
   PRODUCT_TYPE[2].Motion.Gluing_Nozzle_Z.Position[1].Pos := 143.76;
   PRODUCT_TYPE[2].Motion.Gluing_Nozzle_Z.Position[2].Pos := 139.11;
   PRODUCT_TYPE[2].Motion.Gluing_Nozzle_Z.Position[3].Pos := 131.98;
   PRODUCT_TYPE[2].Motion.Gluing_Nozzle_Z.Position[4].Pos := 127.89;
   PRODUCT_TYPE[2].Motion.Gluing_Nozzle_Z.Position[6].Pos := 127.0;
   PRODUCT_TYPE[2].Motion.Gluing_Nozzle_Z.Position[7].Pos := 48.11;
   PRODUCT_TYPE[2].Motion.Gluing_Nozzle_Z.Position[9].Pos := 123.0;
   PRODUCT_TYPE[3].Motion.Gluing_Nozzle_Z.Position[1].Pos := 143.76;
   PRODUCT_TYPE[3].Motion.Gluing_Nozzle_Z.Position[2].Pos := 139.11;
   PRODUCT_TYPE[3].Motion.Gluing_Nozzle_Z.Position[3].Pos := 131.98;
   PRODUCT_TYPE[3].Motion.Gluing_Nozzle_Z.Position[4].Pos := 127.89;
   PRODUCT_TYPE[3].Motion.Gluing_Nozzle_Z.Position[6].Pos := 127.0;
   PRODUCT_TYPE[3].Motion.Gluing_Nozzle_Z.Position[7].Pos := 48.11;
   PRODUCT_TYPE[3].Motion.Gluing_Nozzle_Z.Position[9].Pos := 123.0;
   PRODUCT_TYPE[4].Motion.Gluing_Nozzle_Z.Position[1].Pos := 143.76;
   PRODUCT_TYPE[4].Motion.Gluing_Nozzle_Z.Position[2].Pos := 139.11;
   PRODUCT_TYPE[4].Motion.Gluing_Nozzle_Z.Position[3].Pos := 131.98;
   PRODUCT_TYPE[4].Motion.Gluing_Nozzle_Z.Position[4].Pos := 127.89;
   PRODUCT_TYPE[4].Motion.Gluing_Nozzle_Z.Position[6].Pos := 127.0;
   PRODUCT_TYPE[4].Motion.Gluing_Nozzle_Z.Position[7].Pos := 48.11;
   PRODUCT_TYPE[4].Motion.Gluing_Nozzle_Z.Position[9].Pos := 123.0;
   PRODUCT_TYPE[5].Motion.Gluing_Nozzle_Z.Position[1].Pos := 143.76;
   PRODUCT_TYPE[5].Motion.Gluing_Nozzle_Z.Position[2].Pos := 139.11;
   PRODUCT_TYPE[5].Motion.Gluing_Nozzle_Z.Position[3].Pos := 131.98;
   PRODUCT_TYPE[5].Motion.Gluing_Nozzle_Z.Position[4].Pos := 127.89;
   PRODUCT_TYPE[5].Motion.Gluing_Nozzle_Z.Position[6].Pos := 127.0;
   PRODUCT_TYPE[5].Motion.Gluing_Nozzle_Z.Position[7].Pos := 48.11;
   PRODUCT_TYPE[5].Motion.Gluing_Nozzle_Z.Position[9].Pos := 123.0;
   PRODUCT_TYPE[6].Motion.Gluing_Nozzle_Z.Position[1].Pos := 143.76;
   PRODUCT_TYPE[6].Motion.Gluing_Nozzle_Z.Position[2].Pos := 139.11;
   PRODUCT_TYPE[6].Motion.Gluing_Nozzle_Z.Position[3].Pos := 131.98;
   PRODUCT_TYPE[6].Motion.Gluing_Nozzle_Z.Position[4].Pos := 127.89;
   PRODUCT_TYPE[6].Motion.Gluing_Nozzle_Z.Position[6].Pos := 127.0;
   PRODUCT_TYPE[6].Motion.Gluing_Nozzle_Z.Position[7].Pos := 48.11;
   PRODUCT_TYPE[6].Motion.Gluing_Nozzle_Z.Position[9].Pos := 123.0;
   PRODUCT_TYPE[7].Motion.Gluing_Nozzle_Z.Position[1].Pos := 143.76;
   PRODUCT_TYPE[7].Motion.Gluing_Nozzle_Z.Position[2].Pos := 139.11;
   PRODUCT_TYPE[7].Motion.Gluing_Nozzle_Z.Position[3].Pos := 131.98;
   PRODUCT_TYPE[7].Motion.Gluing_Nozzle_Z.Position[4].Pos := 127.89;
   PRODUCT_TYPE[7].Motion.Gluing_Nozzle_Z.Position[6].Pos := 127.0;
   PRODUCT_TYPE[7].Motion.Gluing_Nozzle_Z.Position[7].Pos := 48.11;
   PRODUCT_TYPE[7].Motion.Gluing_Nozzle_Z.Position[9].Pos := 123.0;
   PRODUCT_TYPE[8].Motion.Gluing_Nozzle_Z.Position[1].Pos := 143.76;
   PRODUCT_TYPE[8].Motion.Gluing_Nozzle_Z.Position[2].Pos := 139.11;
   PRODUCT_TYPE[8].Motion.Gluing_Nozzle_Z.Position[3].Pos := 131.98;
   PRODUCT_TYPE[8].Motion.Gluing_Nozzle_Z.Position[4].Pos := 127.89;
   PRODUCT_TYPE[8].Motion.Gluing_Nozzle_Z.Position[6].Pos := 127.0;
   PRODUCT_TYPE[8].Motion.Gluing_Nozzle_Z.Position[7].Pos := 48.11;
   PRODUCT_TYPE[8].Motion.Gluing_Nozzle_Z.Position[9].Pos := 123.0;
   PRODUCT_TYPE[9].Motion.Gluing_Nozzle_Z.Position[1].Pos := 143.76;
   PRODUCT_TYPE[9].Motion.Gluing_Nozzle_Z.Position[2].Pos := 139.11;
   PRODUCT_TYPE[9].Motion.Gluing_Nozzle_Z.Position[3].Pos := 131.98;
   PRODUCT_TYPE[9].Motion.Gluing_Nozzle_Z.Position[4].Pos := 127.89;
   PRODUCT_TYPE[9].Motion.Gluing_Nozzle_Z.Position[6].Pos := 127.0;
   PRODUCT_TYPE[9].Motion.Gluing_Nozzle_Z.Position[7].Pos := 48.11;
   PRODUCT_TYPE[9].Motion.Gluing_Nozzle_Z.Position[9].Pos := 123.0;
   PRODUCT_TYPE[10].Motion.Gluing_Nozzle_Z.Position[1].Pos := 143.76;
   PRODUCT_TYPE[10].Motion.Gluing_Nozzle_Z.Position[2].Pos := 139.11;
   PRODUCT_TYPE[10].Motion.Gluing_Nozzle_Z.Position[3].Pos := 131.98;
   PRODUCT_TYPE[10].Motion.Gluing_Nozzle_Z.Position[4].Pos := 127.89;
   PRODUCT_TYPE[10].Motion.Gluing_Nozzle_Z.Position[6].Pos := 127.0;
   PRODUCT_TYPE[10].Motion.Gluing_Nozzle_Z.Position[7].Pos := 48.11;
   PRODUCT_TYPE[10].Motion.Gluing_Nozzle_Z.Position[9].Pos := 123.0;
   PRODUCT_TYPE[1].Motion.Gluing_Nozzle_Z.Position[1..4].Vel := 200;
   PRODUCT_TYPE[1].Motion.Gluing_Nozzle_Z.Position[6..9].Vel := 200;
   PRODUCT_TYPE[2].Motion.Gluing_Nozzle_Z.Position[1..4].Vel := 200;
   PRODUCT_TYPE[2].Motion.Gluing_Nozzle_Z.Position[6..9].Vel := 200;
   PRODUCT_TYPE[3].Motion.Gluing_Nozzle_Z.Position[1..4].Vel := 200;
   PRODUCT_TYPE[3].Motion.Gluing_Nozzle_Z.Position[6..9].Vel := 200;
   PRODUCT_TYPE[4].Motion.Gluing_Nozzle_Z.Position[1..4].Vel := 200;
   PRODUCT_TYPE[4].Motion.Gluing_Nozzle_Z.Position[6..9].Vel := 200;
   PRODUCT_TYPE[5].Motion.Gluing_Nozzle_Z.Position[1..4].Vel := 200;
   PRODUCT_TYPE[5].Motion.Gluing_Nozzle_Z.Position[6..9].Vel := 200;
   PRODUCT_TYPE[6].Motion.Gluing_Nozzle_Z.Position[1..4].Vel := 200;
   PRODUCT_TYPE[6].Motion.Gluing_Nozzle_Z.Position[6..9].Vel := 200;
   PRODUCT_TYPE[7].Motion.Gluing_Nozzle_Z.Position[1..4].Vel := 200;
   PRODUCT_TYPE[7].Motion.Gluing_Nozzle_Z.Position[6..9].Vel := 200;
   PRODUCT_TYPE[8].Motion.Gluing_Nozzle_Z.Position[1..4].Vel := 200;
   PRODUCT_TYPE[8].Motion.Gluing_Nozzle_Z.Position[6..9].Vel := 200;
   PRODUCT_TYPE[9].Motion.Gluing_Nozzle_Z.Position[1..4].Vel := 200;
   PRODUCT_TYPE[9].Motion.Gluing_Nozzle_Z.Position[6..9].Vel := 200;
   PRODUCT_TYPE[10].Motion.Gluing_Nozzle_Z.Position[1..4].Vel := 200;
   PRODUCT_TYPE[10].Motion.Gluing_Nozzle_Z.Position[6..9].Vel := 200;
   PRODUCT_TYPE[1].Motion.Gluing_Nozzle_X.Position[1].Pos := 2.34;
   PRODUCT_TYPE[1].Motion.Gluing_Nozzle_X.Position[2].Pos := 76.0;
   PRODUCT_TYPE[1].Motion.Gluing_Nozzle_X.Position[3..6].Pos := 84.69;
   PRODUCT_TYPE[1].Motion.Gluing_Nozzle_X.Position[7].Pos := 85.0;
   PRODUCT_TYPE[1].Motion.Gluing_Nozzle_X.Position[8].Pos := 88.53;
   PRODUCT_TYPE[2].Motion.Gluing_Nozzle_X.Position[1].Pos := 2.34;
   PRODUCT_TYPE[2].Motion.Gluing_Nozzle_X.Position[2].Pos := 76.0;
   PRODUCT_TYPE[2].Motion.Gluing_Nozzle_X.Position[3..6].Pos := 84.69;
   PRODUCT_TYPE[2].Motion.Gluing_Nozzle_X.Position[7].Pos := 85.0;
   PRODUCT_TYPE[2].Motion.Gluing_Nozzle_X.Position[8].Pos := 88.53;
   PRODUCT_TYPE[3].Motion.Gluing_Nozzle_X.Position[1].Pos := 2.34;
   PRODUCT_TYPE[3].Motion.Gluing_Nozzle_X.Position[2].Pos := 76.0;
   PRODUCT_TYPE[3].Motion.Gluing_Nozzle_X.Position[3..6].Pos := 84.69;
   PRODUCT_TYPE[3].Motion.Gluing_Nozzle_X.Position[7].Pos := 85.0;
   PRODUCT_TYPE[3].Motion.Gluing_Nozzle_X.Position[8].Pos := 88.53;
   PRODUCT_TYPE[4].Motion.Gluing_Nozzle_X.Position[1].Pos := 2.34;
   PRODUCT_TYPE[4].Motion.Gluing_Nozzle_X.Position[2].Pos := 76.0;
   PRODUCT_TYPE[4].Motion.Gluing_Nozzle_X.Position[3..6].Pos := 84.69;
   PRODUCT_TYPE[4].Motion.Gluing_Nozzle_X.Position[7].Pos := 85.0;
   PRODUCT_TYPE[4].Motion.Gluing_Nozzle_X.Position[8].Pos := 88.53;
   PRODUCT_TYPE[5].Motion.Gluing_Nozzle_X.Position[1].Pos := 2.34;
   PRODUCT_TYPE[5].Motion.Gluing_Nozzle_X.Position[2].Pos := 76.0;
   PRODUCT_TYPE[5].Motion.Gluing_Nozzle_X.Position[3..6].Pos := 84.69;
   PRODUCT_TYPE[5].Motion.Gluing_Nozzle_X.Position[7].Pos := 85.0;
   PRODUCT_TYPE[5].Motion.Gluing_Nozzle_X.Position[8].Pos := 88.53;
   PRODUCT_TYPE[6].Motion.Gluing_Nozzle_X.Position[1].Pos := 2.34;
   PRODUCT_TYPE[6].Motion.Gluing_Nozzle_X.Position[2].Pos := 76.0;
   PRODUCT_TYPE[6].Motion.Gluing_Nozzle_X.Position[3..6].Pos := 84.69;
   PRODUCT_TYPE[6].Motion.Gluing_Nozzle_X.Position[7].Pos := 85.0;
   PRODUCT_TYPE[6].Motion.Gluing_Nozzle_X.Position[8].Pos := 88.53;
   PRODUCT_TYPE[7].Motion.Gluing_Nozzle_X.Position[1].Pos := 2.34;
   PRODUCT_TYPE[7].Motion.Gluing_Nozzle_X.Position[2].Pos := 76.0;
   PRODUCT_TYPE[7].Motion.Gluing_Nozzle_X.Position[3..6].Pos := 84.69;
   PRODUCT_TYPE[7].Motion.Gluing_Nozzle_X.Position[7].Pos := 85.0;
   PRODUCT_TYPE[7].Motion.Gluing_Nozzle_X.Position[8].Pos := 88.53;
   PRODUCT_TYPE[8].Motion.Gluing_Nozzle_X.Position[1].Pos := 2.34;
   PRODUCT_TYPE[8].Motion.Gluing_Nozzle_X.Position[2].Pos := 76.0;
   PRODUCT_TYPE[8].Motion.Gluing_Nozzle_X.Position[3..6].Pos := 84.69;
   PRODUCT_TYPE[8].Motion.Gluing_Nozzle_X.Position[7].Pos := 85.0;
   PRODUCT_TYPE[8].Motion.Gluing_Nozzle_X.Position[8].Pos := 88.53;
   PRODUCT_TYPE[9].Motion.Gluing_Nozzle_X.Position[1].Pos := 2.34;
   PRODUCT_TYPE[9].Motion.Gluing_Nozzle_X.Position[2].Pos := 76.0;
   PRODUCT_TYPE[9].Motion.Gluing_Nozzle_X.Position[3..6].Pos := 84.69;
   PRODUCT_TYPE[9].Motion.Gluing_Nozzle_X.Position[7].Pos := 85.0;
   PRODUCT_TYPE[9].Motion.Gluing_Nozzle_X.Position[8].Pos := 88.53;
   PRODUCT_TYPE[10].Motion.Gluing_Nozzle_X.Position[1].Pos := 2.34;
   PRODUCT_TYPE[10].Motion.Gluing_Nozzle_X.Position[2].Pos := 76.0;
   PRODUCT_TYPE[10].Motion.Gluing_Nozzle_X.Position[3..6].Pos := 84.69;
   PRODUCT_TYPE[10].Motion.Gluing_Nozzle_X.Position[7].Pos := 85.0;
   PRODUCT_TYPE[10].Motion.Gluing_Nozzle_X.Position[8].Pos := 88.53;
   PRODUCT_TYPE[1].Motion.Gluing_Nozzle_X.Position[1..8].Vel := 200;
   PRODUCT_TYPE[2].Motion.Gluing_Nozzle_X.Position[1..8].Vel := 200;
   PRODUCT_TYPE[3].Motion.Gluing_Nozzle_X.Position[1..8].Vel := 200;
   PRODUCT_TYPE[4].Motion.Gluing_Nozzle_X.Position[1..8].Vel := 200;
   PRODUCT_TYPE[5].Motion.Gluing_Nozzle_X.Position[1..8].Vel := 200;
   PRODUCT_TYPE[6].Motion.Gluing_Nozzle_X.Position[1..8].Vel := 200;
   PRODUCT_TYPE[7].Motion.Gluing_Nozzle_X.Position[1..8].Vel := 200;
   PRODUCT_TYPE[8].Motion.Gluing_Nozzle_X.Position[1..8].Vel := 200;
   PRODUCT_TYPE[9].Motion.Gluing_Nozzle_X.Position[1..8].Vel := 200;
   PRODUCT_TYPE[10].Motion.Gluing_Nozzle_X.Position[1..8].Vel := 200;
   PRODUCT_TYPE[1].Motion.Gluing_Nozzle_Y.Position[1..5].Pos := 115.47;
   PRODUCT_TYPE[1].Motion.Gluing_Nozzle_Y.Position[6].Pos := 110.18;
   PRODUCT_TYPE[1].Motion.Gluing_Nozzle_Y.Position[7].Pos := 60.52;
   PRODUCT_TYPE[1].Motion.Gluing_Nozzle_Y.Position[8].Pos := 80.0;
   PRODUCT_TYPE[2].Motion.Gluing_Nozzle_Y.Position[1..5].Pos := 115.47;
   PRODUCT_TYPE[2].Motion.Gluing_Nozzle_Y.Position[6].Pos := 110.18;
   PRODUCT_TYPE[2].Motion.Gluing_Nozzle_Y.Position[7].Pos := 60.52;
   PRODUCT_TYPE[2].Motion.Gluing_Nozzle_Y.Position[8].Pos := 80.0;
   PRODUCT_TYPE[3].Motion.Gluing_Nozzle_Y.Position[1..5].Pos := 115.47;
   PRODUCT_TYPE[3].Motion.Gluing_Nozzle_Y.Position[6].Pos := 110.18;
   PRODUCT_TYPE[3].Motion.Gluing_Nozzle_Y.Position[7].Pos := 60.52;
   PRODUCT_TYPE[3].Motion.Gluing_Nozzle_Y.Position[8].Pos := 80.0;
   PRODUCT_TYPE[4].Motion.Gluing_Nozzle_Y.Position[1..5].Pos := 115.47;
   PRODUCT_TYPE[4].Motion.Gluing_Nozzle_Y.Position[6].Pos := 110.18;
   PRODUCT_TYPE[4].Motion.Gluing_Nozzle_Y.Position[7].Pos := 60.52;
   PRODUCT_TYPE[4].Motion.Gluing_Nozzle_Y.Position[8].Pos := 80.0;
   PRODUCT_TYPE[5].Motion.Gluing_Nozzle_Y.Position[1..5].Pos := 115.47;
   PRODUCT_TYPE[5].Motion.Gluing_Nozzle_Y.Position[6].Pos := 110.18;
   PRODUCT_TYPE[5].Motion.Gluing_Nozzle_Y.Position[7].Pos := 60.52;
   PRODUCT_TYPE[5].Motion.Gluing_Nozzle_Y.Position[8].Pos := 80.0;
   PRODUCT_TYPE[6].Motion.Gluing_Nozzle_Y.Position[1..5].Pos := 115.47;
   PRODUCT_TYPE[6].Motion.Gluing_Nozzle_Y.Position[6].Pos := 110.18;
   PRODUCT_TYPE[6].Motion.Gluing_Nozzle_Y.Position[7].Pos := 60.52;
   PRODUCT_TYPE[6].Motion.Gluing_Nozzle_Y.Position[8].Pos := 80.0;
   PRODUCT_TYPE[7].Motion.Gluing_Nozzle_Y.Position[1..5].Pos := 115.47;
   PRODUCT_TYPE[7].Motion.Gluing_Nozzle_Y.Position[6].Pos := 110.18;
   PRODUCT_TYPE[7].Motion.Gluing_Nozzle_Y.Position[7].Pos := 60.52;
   PRODUCT_TYPE[7].Motion.Gluing_Nozzle_Y.Position[8].Pos := 80.0;
   PRODUCT_TYPE[8].Motion.Gluing_Nozzle_Y.Position[1..5].Pos := 115.47;
   PRODUCT_TYPE[8].Motion.Gluing_Nozzle_Y.Position[6].Pos := 110.18;
   PRODUCT_TYPE[8].Motion.Gluing_Nozzle_Y.Position[7].Pos := 60.52;
   PRODUCT_TYPE[8].Motion.Gluing_Nozzle_Y.Position[8].Pos := 80.0;
   PRODUCT_TYPE[9].Motion.Gluing_Nozzle_Y.Position[1..5].Pos := 115.47;
   PRODUCT_TYPE[9].Motion.Gluing_Nozzle_Y.Position[6].Pos := 110.18;
   PRODUCT_TYPE[9].Motion.Gluing_Nozzle_Y.Position[7].Pos := 60.52;
   PRODUCT_TYPE[9].Motion.Gluing_Nozzle_Y.Position[8].Pos := 80.0;
   PRODUCT_TYPE[10].Motion.Gluing_Nozzle_Y.Position[1..5].Pos := 115.47;
   PRODUCT_TYPE[10].Motion.Gluing_Nozzle_Y.Position[6].Pos := 110.18;
   PRODUCT_TYPE[10].Motion.Gluing_Nozzle_Y.Position[7].Pos := 60.52;
   PRODUCT_TYPE[10].Motion.Gluing_Nozzle_Y.Position[8].Pos := 80.0;
   PRODUCT_TYPE[1].Motion.Gluing_Nozzle_Y.Position[1..7].Vel := 200;
   PRODUCT_TYPE[1].Motion.Gluing_Nozzle_Y.Position[8].Vel := 100;
   PRODUCT_TYPE[2].Motion.Gluing_Nozzle_Y.Position[1..7].Vel := 200;
   PRODUCT_TYPE[2].Motion.Gluing_Nozzle_Y.Position[8].Vel := 100;
   PRODUCT_TYPE[3].Motion.Gluing_Nozzle_Y.Position[1..7].Vel := 200;
   PRODUCT_TYPE[3].Motion.Gluing_Nozzle_Y.Position[8].Vel := 100;
   PRODUCT_TYPE[4].Motion.Gluing_Nozzle_Y.Position[1..7].Vel := 200;
   PRODUCT_TYPE[4].Motion.Gluing_Nozzle_Y.Position[8].Vel := 100;
   PRODUCT_TYPE[5].Motion.Gluing_Nozzle_Y.Position[1..7].Vel := 200;
   PRODUCT_TYPE[5].Motion.Gluing_Nozzle_Y.Position[8].Vel := 100;
   PRODUCT_TYPE[6].Motion.Gluing_Nozzle_Y.Position[1..7].Vel := 200;
   PRODUCT_TYPE[6].Motion.Gluing_Nozzle_Y.Position[8].Vel := 100;
   PRODUCT_TYPE[7].Motion.Gluing_Nozzle_Y.Position[1..7].Vel := 200;
   PRODUCT_TYPE[7].Motion.Gluing_Nozzle_Y.Position[8].Vel := 100;
   PRODUCT_TYPE[8].Motion.Gluing_Nozzle_Y.Position[1..7].Vel := 200;
   PRODUCT_TYPE[8].Motion.Gluing_Nozzle_Y.Position[8].Vel := 100;
   PRODUCT_TYPE[9].Motion.Gluing_Nozzle_Y.Position[1..7].Vel := 200;
   PRODUCT_TYPE[9].Motion.Gluing_Nozzle_Y.Position[8].Vel := 100;
   PRODUCT_TYPE[10].Motion.Gluing_Nozzle_Y.Position[1..7].Vel := 200;
   PRODUCT_TYPE[10].Motion.Gluing_Nozzle_Y.Position[8].Vel := 100;
   PRODUCT_TYPE[1].Motion.Ring_Turntable_Axis_1.Position[1].Pos := 3419;
   PRODUCT_TYPE[1].Motion.Ring_Turntable_Axis_1.Position[2].Pos := 48386;
   PRODUCT_TYPE[1].Motion.Ring_Turntable_Axis_1.Position[3].Pos := 93294;
   PRODUCT_TYPE[1].Motion.Ring_Turntable_Axis_1.Position[4].Pos := 138335;
   PRODUCT_TYPE[1].Motion.Ring_Turntable_Axis_1.Position[5].Pos := 183464;
   PRODUCT_TYPE[1].Motion.Ring_Turntable_Axis_1.Position[6].Pos := 228443;
   PRODUCT_TYPE[1].Motion.Ring_Turntable_Axis_1.Position[7].Pos := 273535;
   PRODUCT_TYPE[1].Motion.Ring_Turntable_Axis_1.Position[8].Pos := 318250;
   PRODUCT_TYPE[2].Motion.Ring_Turntable_Axis_1.Position[1].Pos := 3419;
   PRODUCT_TYPE[2].Motion.Ring_Turntable_Axis_1.Position[2].Pos := 48386;
   PRODUCT_TYPE[2].Motion.Ring_Turntable_Axis_1.Position[3].Pos := 93294;
   PRODUCT_TYPE[2].Motion.Ring_Turntable_Axis_1.Position[4].Pos := 138335;
   PRODUCT_TYPE[2].Motion.Ring_Turntable_Axis_1.Position[5].Pos := 183464;
   PRODUCT_TYPE[2].Motion.Ring_Turntable_Axis_1.Position[6].Pos := 228443;
   PRODUCT_TYPE[2].Motion.Ring_Turntable_Axis_1.Position[7].Pos := 273535;
   PRODUCT_TYPE[2].Motion.Ring_Turntable_Axis_1.Position[8].Pos := 318250;
   PRODUCT_TYPE[3].Motion.Ring_Turntable_Axis_1.Position[1].Pos := 3419;
   PRODUCT_TYPE[3].Motion.Ring_Turntable_Axis_1.Position[2].Pos := 48386;
   PRODUCT_TYPE[3].Motion.Ring_Turntable_Axis_1.Position[3].Pos := 93294;
   PRODUCT_TYPE[3].Motion.Ring_Turntable_Axis_1.Position[4].Pos := 138335;
   PRODUCT_TYPE[3].Motion.Ring_Turntable_Axis_1.Position[5].Pos := 183464;
   PRODUCT_TYPE[3].Motion.Ring_Turntable_Axis_1.Position[6].Pos := 228443;
   PRODUCT_TYPE[3].Motion.Ring_Turntable_Axis_1.Position[7].Pos := 273535;
   PRODUCT_TYPE[3].Motion.Ring_Turntable_Axis_1.Position[8].Pos := 318250;
   PRODUCT_TYPE[4].Motion.Ring_Turntable_Axis_1.Position[1].Pos := 3419;
   PRODUCT_TYPE[4].Motion.Ring_Turntable_Axis_1.Position[2].Pos := 48386;
   PRODUCT_TYPE[4].Motion.Ring_Turntable_Axis_1.Position[3].Pos := 93294;
   PRODUCT_TYPE[4].Motion.Ring_Turntable_Axis_1.Position[4].Pos := 138335;
   PRODUCT_TYPE[4].Motion.Ring_Turntable_Axis_1.Position[5].Pos := 183464;
   PRODUCT_TYPE[4].Motion.Ring_Turntable_Axis_1.Position[6].Pos := 228443;
   PRODUCT_TYPE[4].Motion.Ring_Turntable_Axis_1.Position[7].Pos := 273535;
   PRODUCT_TYPE[4].Motion.Ring_Turntable_Axis_1.Position[8].Pos := 318250;
   PRODUCT_TYPE[5].Motion.Ring_Turntable_Axis_1.Position[1].Pos := 3419;
   PRODUCT_TYPE[5].Motion.Ring_Turntable_Axis_1.Position[2].Pos := 48386;
   PRODUCT_TYPE[5].Motion.Ring_Turntable_Axis_1.Position[3].Pos := 93294;
   PRODUCT_TYPE[5].Motion.Ring_Turntable_Axis_1.Position[4].Pos := 138335;
   PRODUCT_TYPE[5].Motion.Ring_Turntable_Axis_1.Position[5].Pos := 183464;
   PRODUCT_TYPE[5].Motion.Ring_Turntable_Axis_1.Position[6].Pos := 228443;
   PRODUCT_TYPE[5].Motion.Ring_Turntable_Axis_1.Position[7].Pos := 273535;
   PRODUCT_TYPE[5].Motion.Ring_Turntable_Axis_1.Position[8].Pos := 318250;
   PRODUCT_TYPE[6].Motion.Ring_Turntable_Axis_1.Position[1].Pos := 3419;
   PRODUCT_TYPE[6].Motion.Ring_Turntable_Axis_1.Position[2].Pos := 48386;
   PRODUCT_TYPE[6].Motion.Ring_Turntable_Axis_1.Position[3].Pos := 93294;
   PRODUCT_TYPE[6].Motion.Ring_Turntable_Axis_1.Position[4].Pos := 138335;
   PRODUCT_TYPE[6].Motion.Ring_Turntable_Axis_1.Position[5].Pos := 183464;
   PRODUCT_TYPE[6].Motion.Ring_Turntable_Axis_1.Position[6].Pos := 228443;
   PRODUCT_TYPE[6].Motion.Ring_Turntable_Axis_1.Position[7].Pos := 273535;
   PRODUCT_TYPE[6].Motion.Ring_Turntable_Axis_1.Position[8].Pos := 318250;
   PRODUCT_TYPE[7].Motion.Ring_Turntable_Axis_1.Position[1].Pos := 3419;
   PRODUCT_TYPE[7].Motion.Ring_Turntable_Axis_1.Position[2].Pos := 48386;
   PRODUCT_TYPE[7].Motion.Ring_Turntable_Axis_1.Position[3].Pos := 93294;
   PRODUCT_TYPE[7].Motion.Ring_Turntable_Axis_1.Position[4].Pos := 138335;
   PRODUCT_TYPE[7].Motion.Ring_Turntable_Axis_1.Position[5].Pos := 183464;
   PRODUCT_TYPE[7].Motion.Ring_Turntable_Axis_1.Position[6].Pos := 228443;
   PRODUCT_TYPE[7].Motion.Ring_Turntable_Axis_1.Position[7].Pos := 273535;
   PRODUCT_TYPE[7].Motion.Ring_Turntable_Axis_1.Position[8].Pos := 318250;
   PRODUCT_TYPE[8].Motion.Ring_Turntable_Axis_1.Position[1].Pos := 3419;
   PRODUCT_TYPE[8].Motion.Ring_Turntable_Axis_1.Position[2].Pos := 48386;
   PRODUCT_TYPE[8].Motion.Ring_Turntable_Axis_1.Position[3].Pos := 93294;
   PRODUCT_TYPE[8].Motion.Ring_Turntable_Axis_1.Position[4].Pos := 138335;
   PRODUCT_TYPE[8].Motion.Ring_Turntable_Axis_1.Position[5].Pos := 183464;
   PRODUCT_TYPE[8].Motion.Ring_Turntable_Axis_1.Position[6].Pos := 228443;
   PRODUCT_TYPE[8].Motion.Ring_Turntable_Axis_1.Position[7].Pos := 273535;
   PRODUCT_TYPE[8].Motion.Ring_Turntable_Axis_1.Position[8].Pos := 318250;
   PRODUCT_TYPE[9].Motion.Ring_Turntable_Axis_1.Position[1].Pos := 3419;
   PRODUCT_TYPE[9].Motion.Ring_Turntable_Axis_1.Position[2].Pos := 48386;
   PRODUCT_TYPE[9].Motion.Ring_Turntable_Axis_1.Position[3].Pos := 93294;
   PRODUCT_TYPE[9].Motion.Ring_Turntable_Axis_1.Position[4].Pos := 138335;
   PRODUCT_TYPE[9].Motion.Ring_Turntable_Axis_1.Position[5].Pos := 183464;
   PRODUCT_TYPE[9].Motion.Ring_Turntable_Axis_1.Position[6].Pos := 228443;
   PRODUCT_TYPE[9].Motion.Ring_Turntable_Axis_1.Position[7].Pos := 273535;
   PRODUCT_TYPE[9].Motion.Ring_Turntable_Axis_1.Position[8].Pos := 318250;
   PRODUCT_TYPE[10].Motion.Ring_Turntable_Axis_1.Position[1].Pos := 3419;
   PRODUCT_TYPE[10].Motion.Ring_Turntable_Axis_1.Position[2].Pos := 48386;
   PRODUCT_TYPE[10].Motion.Ring_Turntable_Axis_1.Position[3].Pos := 93294;
   PRODUCT_TYPE[10].Motion.Ring_Turntable_Axis_1.Position[4].Pos := 138335;
   PRODUCT_TYPE[10].Motion.Ring_Turntable_Axis_1.Position[5].Pos := 183464;
   PRODUCT_TYPE[10].Motion.Ring_Turntable_Axis_1.Position[6].Pos := 228443;
   PRODUCT_TYPE[10].Motion.Ring_Turntable_Axis_1.Position[7].Pos := 273535;
   PRODUCT_TYPE[10].Motion.Ring_Turntable_Axis_1.Position[8].Pos := 318250;
   PRODUCT_TYPE[1].Motion.Ring_Turntable_Axis_1.Position[1..8].Vel := 10000;
   PRODUCT_TYPE[2].Motion.Ring_Turntable_Axis_1.Position[1..8].Vel := 10000;
   PRODUCT_TYPE[3].Motion.Ring_Turntable_Axis_1.Position[1..8].Vel := 10000;
   PRODUCT_TYPE[4].Motion.Ring_Turntable_Axis_1.Position[1..8].Vel := 10000;
   PRODUCT_TYPE[5].Motion.Ring_Turntable_Axis_1.Position[1..8].Vel := 10000;
   PRODUCT_TYPE[6].Motion.Ring_Turntable_Axis_1.Position[1..8].Vel := 10000;
   PRODUCT_TYPE[7].Motion.Ring_Turntable_Axis_1.Position[1..8].Vel := 10000;
   PRODUCT_TYPE[8].Motion.Ring_Turntable_Axis_1.Position[1..8].Vel := 10000;
   PRODUCT_TYPE[9].Motion.Ring_Turntable_Axis_1.Position[1..8].Vel := 10000;
   PRODUCT_TYPE[10].Motion.Ring_Turntable_Axis_1.Position[1..8].Vel := 10000;
   PRODUCT_TYPE[1].Motion.Shaft_Scan_Turntable_Axis.Position[2].Pos := 450000;
   PRODUCT_TYPE[1].Motion.Shaft_Scan_Turntable_Axis.Position[3].Pos := 900000;
   PRODUCT_TYPE[1].Motion.Shaft_Scan_Turntable_Axis.Position[4].Pos := 135000;
   PRODUCT_TYPE[1].Motion.Shaft_Scan_Turntable_Axis.Position[5].Pos := 180000;
   PRODUCT_TYPE[1].Motion.Shaft_Scan_Turntable_Axis.Position[6].Pos := 225000;
   PRODUCT_TYPE[1].Motion.Shaft_Scan_Turntable_Axis.Position[7].Pos := 270000;
   PRODUCT_TYPE[1].Motion.Shaft_Scan_Turntable_Axis.Position[8].Pos := 315000;
   PRODUCT_TYPE[2].Motion.Shaft_Scan_Turntable_Axis.Position[2].Pos := 450000;
   PRODUCT_TYPE[2].Motion.Shaft_Scan_Turntable_Axis.Position[3].Pos := 900000;
   PRODUCT_TYPE[2].Motion.Shaft_Scan_Turntable_Axis.Position[4].Pos := 135000;
   PRODUCT_TYPE[2].Motion.Shaft_Scan_Turntable_Axis.Position[5].Pos := 180000;
   PRODUCT_TYPE[2].Motion.Shaft_Scan_Turntable_Axis.Position[6].Pos := 225000;
   PRODUCT_TYPE[2].Motion.Shaft_Scan_Turntable_Axis.Position[7].Pos := 270000;
   PRODUCT_TYPE[2].Motion.Shaft_Scan_Turntable_Axis.Position[8].Pos := 315000;
   PRODUCT_TYPE[3].Motion.Shaft_Scan_Turntable_Axis.Position[2].Pos := 450000;
   PRODUCT_TYPE[3].Motion.Shaft_Scan_Turntable_Axis.Position[3].Pos := 900000;
   PRODUCT_TYPE[3].Motion.Shaft_Scan_Turntable_Axis.Position[4].Pos := 135000;
   PRODUCT_TYPE[3].Motion.Shaft_Scan_Turntable_Axis.Position[5].Pos := 180000;
   PRODUCT_TYPE[3].Motion.Shaft_Scan_Turntable_Axis.Position[6].Pos := 225000;
   PRODUCT_TYPE[3].Motion.Shaft_Scan_Turntable_Axis.Position[7].Pos := 270000;
   PRODUCT_TYPE[3].Motion.Shaft_Scan_Turntable_Axis.Position[8].Pos := 315000;
   PRODUCT_TYPE[4].Motion.Shaft_Scan_Turntable_Axis.Position[2].Pos := 450000;
   PRODUCT_TYPE[4].Motion.Shaft_Scan_Turntable_Axis.Position[3].Pos := 900000;
   PRODUCT_TYPE[4].Motion.Shaft_Scan_Turntable_Axis.Position[4].Pos := 135000;
   PRODUCT_TYPE[4].Motion.Shaft_Scan_Turntable_Axis.Position[5].Pos := 180000;
   PRODUCT_TYPE[4].Motion.Shaft_Scan_Turntable_Axis.Position[6].Pos := 225000;
   PRODUCT_TYPE[4].Motion.Shaft_Scan_Turntable_Axis.Position[7].Pos := 270000;
   PRODUCT_TYPE[4].Motion.Shaft_Scan_Turntable_Axis.Position[8].Pos := 315000;
   PRODUCT_TYPE[5].Motion.Shaft_Scan_Turntable_Axis.Position[2].Pos := 450000;
   PRODUCT_TYPE[5].Motion.Shaft_Scan_Turntable_Axis.Position[3].Pos := 900000;
   PRODUCT_TYPE[5].Motion.Shaft_Scan_Turntable_Axis.Position[4].Pos := 135000;
   PRODUCT_TYPE[5].Motion.Shaft_Scan_Turntable_Axis.Position[5].Pos := 180000;
   PRODUCT_TYPE[5].Motion.Shaft_Scan_Turntable_Axis.Position[6].Pos := 225000;
   PRODUCT_TYPE[5].Motion.Shaft_Scan_Turntable_Axis.Position[7].Pos := 270000;
   PRODUCT_TYPE[5].Motion.Shaft_Scan_Turntable_Axis.Position[8].Pos := 315000;
   PRODUCT_TYPE[6].Motion.Shaft_Scan_Turntable_Axis.Position[2].Pos := 450000;
   PRODUCT_TYPE[6].Motion.Shaft_Scan_Turntable_Axis.Position[3].Pos := 900000;
   PRODUCT_TYPE[6].Motion.Shaft_Scan_Turntable_Axis.Position[4].Pos := 135000;
   PRODUCT_TYPE[6].Motion.Shaft_Scan_Turntable_Axis.Position[5].Pos := 180000;
   PRODUCT_TYPE[6].Motion.Shaft_Scan_Turntable_Axis.Position[6].Pos := 225000;
   PRODUCT_TYPE[6].Motion.Shaft_Scan_Turntable_Axis.Position[7].Pos := 270000;
   PRODUCT_TYPE[6].Motion.Shaft_Scan_Turntable_Axis.Position[8].Pos := 315000;
   PRODUCT_TYPE[7].Motion.Shaft_Scan_Turntable_Axis.Position[2].Pos := 450000;
   PRODUCT_TYPE[7].Motion.Shaft_Scan_Turntable_Axis.Position[3].Pos := 900000;
   PRODUCT_TYPE[7].Motion.Shaft_Scan_Turntable_Axis.Position[4].Pos := 135000;
   PRODUCT_TYPE[7].Motion.Shaft_Scan_Turntable_Axis.Position[5].Pos := 180000;
   PRODUCT_TYPE[7].Motion.Shaft_Scan_Turntable_Axis.Position[6].Pos := 225000;
   PRODUCT_TYPE[7].Motion.Shaft_Scan_Turntable_Axis.Position[7].Pos := 270000;
   PRODUCT_TYPE[7].Motion.Shaft_Scan_Turntable_Axis.Position[8].Pos := 315000;
   PRODUCT_TYPE[8].Motion.Shaft_Scan_Turntable_Axis.Position[2].Pos := 450000;
   PRODUCT_TYPE[8].Motion.Shaft_Scan_Turntable_Axis.Position[3].Pos := 900000;
   PRODUCT_TYPE[8].Motion.Shaft_Scan_Turntable_Axis.Position[4].Pos := 135000;
   PRODUCT_TYPE[8].Motion.Shaft_Scan_Turntable_Axis.Position[5].Pos := 180000;
   PRODUCT_TYPE[8].Motion.Shaft_Scan_Turntable_Axis.Position[6].Pos := 225000;
   PRODUCT_TYPE[8].Motion.Shaft_Scan_Turntable_Axis.Position[7].Pos := 270000;
   PRODUCT_TYPE[8].Motion.Shaft_Scan_Turntable_Axis.Position[8].Pos := 315000;
   PRODUCT_TYPE[9].Motion.Shaft_Scan_Turntable_Axis.Position[2].Pos := 450000;
   PRODUCT_TYPE[9].Motion.Shaft_Scan_Turntable_Axis.Position[3].Pos := 900000;
   PRODUCT_TYPE[9].Motion.Shaft_Scan_Turntable_Axis.Position[4].Pos := 135000;
   PRODUCT_TYPE[9].Motion.Shaft_Scan_Turntable_Axis.Position[5].Pos := 180000;
   PRODUCT_TYPE[9].Motion.Shaft_Scan_Turntable_Axis.Position[6].Pos := 225000;
   PRODUCT_TYPE[9].Motion.Shaft_Scan_Turntable_Axis.Position[7].Pos := 270000;
   PRODUCT_TYPE[9].Motion.Shaft_Scan_Turntable_Axis.Position[8].Pos := 315000;
   PRODUCT_TYPE[10].Motion.Shaft_Scan_Turntable_Axis.Position[2].Pos := 450000;
   PRODUCT_TYPE[10].Motion.Shaft_Scan_Turntable_Axis.Position[3].Pos := 900000;
   PRODUCT_TYPE[10].Motion.Shaft_Scan_Turntable_Axis.Position[4].Pos := 135000;
   PRODUCT_TYPE[10].Motion.Shaft_Scan_Turntable_Axis.Position[5].Pos := 180000;
   PRODUCT_TYPE[10].Motion.Shaft_Scan_Turntable_Axis.Position[6].Pos := 225000;
   PRODUCT_TYPE[10].Motion.Shaft_Scan_Turntable_Axis.Position[7].Pos := 270000;
   PRODUCT_TYPE[10].Motion.Shaft_Scan_Turntable_Axis.Position[8].Pos := 315000;
   PRODUCT_TYPE[1].Motion.Shaft_Scan_Turntable_Axis.Position[1..8].Vel := 10000;
   PRODUCT_TYPE[2].Motion.Shaft_Scan_Turntable_Axis.Position[1..8].Vel := 10000;
   PRODUCT_TYPE[3].Motion.Shaft_Scan_Turntable_Axis.Position[1..8].Vel := 10000;
   PRODUCT_TYPE[4].Motion.Shaft_Scan_Turntable_Axis.Position[1..8].Vel := 10000;
   PRODUCT_TYPE[5].Motion.Shaft_Scan_Turntable_Axis.Position[1..8].Vel := 10000;
   PRODUCT_TYPE[6].Motion.Shaft_Scan_Turntable_Axis.Position[1..8].Vel := 10000;
   PRODUCT_TYPE[7].Motion.Shaft_Scan_Turntable_Axis.Position[1..8].Vel := 10000;
   PRODUCT_TYPE[8].Motion.Shaft_Scan_Turntable_Axis.Position[1..8].Vel := 10000;
   PRODUCT_TYPE[9].Motion.Shaft_Scan_Turntable_Axis.Position[1..8].Vel := 10000;
   PRODUCT_TYPE[10].Motion.Shaft_Scan_Turntable_Axis.Position[1..8].Vel := 10000;
   PRODUCT_TYPE[1].Motion.Gluing_Rotary_Jig_Axis.Position[3..6].Pos := 680000;
   PRODUCT_TYPE[1].Motion.Gluing_Rotary_Jig_Axis.Position[7].Pos := 90000;
   PRODUCT_TYPE[1].Motion.Gluing_Rotary_Jig_Axis.Position[8].Pos := 180000;
   PRODUCT_TYPE[1].Motion.Gluing_Rotary_Jig_Axis.Position[9].Pos := 270000;
   PRODUCT_TYPE[2].Motion.Gluing_Rotary_Jig_Axis.Position[3..6].Pos := 680000;
   PRODUCT_TYPE[2].Motion.Gluing_Rotary_Jig_Axis.Position[7].Pos := 90000;
   PRODUCT_TYPE[2].Motion.Gluing_Rotary_Jig_Axis.Position[8].Pos := 180000;
   PRODUCT_TYPE[2].Motion.Gluing_Rotary_Jig_Axis.Position[9].Pos := 270000;
   PRODUCT_TYPE[3].Motion.Gluing_Rotary_Jig_Axis.Position[3..6].Pos := 680000;
   PRODUCT_TYPE[3].Motion.Gluing_Rotary_Jig_Axis.Position[7].Pos := 90000;
   PRODUCT_TYPE[3].Motion.Gluing_Rotary_Jig_Axis.Position[8].Pos := 180000;
   PRODUCT_TYPE[3].Motion.Gluing_Rotary_Jig_Axis.Position[9].Pos := 270000;
   PRODUCT_TYPE[4].Motion.Gluing_Rotary_Jig_Axis.Position[3..6].Pos := 680000;
   PRODUCT_TYPE[4].Motion.Gluing_Rotary_Jig_Axis.Position[7].Pos := 90000;
   PRODUCT_TYPE[4].Motion.Gluing_Rotary_Jig_Axis.Position[8].Pos := 180000;
   PRODUCT_TYPE[4].Motion.Gluing_Rotary_Jig_Axis.Position[9].Pos := 270000;
   PRODUCT_TYPE[5].Motion.Gluing_Rotary_Jig_Axis.Position[3..6].Pos := 680000;
   PRODUCT_TYPE[5].Motion.Gluing_Rotary_Jig_Axis.Position[7].Pos := 90000;
   PRODUCT_TYPE[5].Motion.Gluing_Rotary_Jig_Axis.Position[8].Pos := 180000;
   PRODUCT_TYPE[5].Motion.Gluing_Rotary_Jig_Axis.Position[9].Pos := 270000;
   PRODUCT_TYPE[6].Motion.Gluing_Rotary_Jig_Axis.Position[3..6].Pos := 680000;
   PRODUCT_TYPE[6].Motion.Gluing_Rotary_Jig_Axis.Position[7].Pos := 90000;
   PRODUCT_TYPE[6].Motion.Gluing_Rotary_Jig_Axis.Position[8].Pos := 180000;
   PRODUCT_TYPE[6].Motion.Gluing_Rotary_Jig_Axis.Position[9].Pos := 270000;
   PRODUCT_TYPE[7].Motion.Gluing_Rotary_Jig_Axis.Position[3..6].Pos := 680000;
   PRODUCT_TYPE[7].Motion.Gluing_Rotary_Jig_Axis.Position[7].Pos := 90000;
   PRODUCT_TYPE[7].Motion.Gluing_Rotary_Jig_Axis.Position[8].Pos := 180000;
   PRODUCT_TYPE[7].Motion.Gluing_Rotary_Jig_Axis.Position[9].Pos := 270000;
   PRODUCT_TYPE[8].Motion.Gluing_Rotary_Jig_Axis.Position[3..6].Pos := 680000;
   PRODUCT_TYPE[8].Motion.Gluing_Rotary_Jig_Axis.Position[7].Pos := 90000;
   PRODUCT_TYPE[8].Motion.Gluing_Rotary_Jig_Axis.Position[8].Pos := 180000;
   PRODUCT_TYPE[8].Motion.Gluing_Rotary_Jig_Axis.Position[9].Pos := 270000;
   PRODUCT_TYPE[9].Motion.Gluing_Rotary_Jig_Axis.Position[3..6].Pos := 680000;
   PRODUCT_TYPE[9].Motion.Gluing_Rotary_Jig_Axis.Position[7].Pos := 90000;
   PRODUCT_TYPE[9].Motion.Gluing_Rotary_Jig_Axis.Position[8].Pos := 180000;
   PRODUCT_TYPE[9].Motion.Gluing_Rotary_Jig_Axis.Position[9].Pos := 270000;
   PRODUCT_TYPE[10].Motion.Gluing_Rotary_Jig_Axis.Position[3..6].Pos := 680000;
   PRODUCT_TYPE[10].Motion.Gluing_Rotary_Jig_Axis.Position[7].Pos := 90000;
   PRODUCT_TYPE[10].Motion.Gluing_Rotary_Jig_Axis.Position[8].Pos := 180000;
   PRODUCT_TYPE[10].Motion.Gluing_Rotary_Jig_Axis.Position[9].Pos := 270000;
   PRODUCT_TYPE[1].Motion.Gluing_Rotary_Jig_Axis.Position[1..2].Vel := 20000;
   PRODUCT_TYPE[1].Motion.Gluing_Rotary_Jig_Axis.Position[3..9].Vel := 10000;
   PRODUCT_TYPE[2].Motion.Gluing_Rotary_Jig_Axis.Position[1..2].Vel := 20000;
   PRODUCT_TYPE[2].Motion.Gluing_Rotary_Jig_Axis.Position[3..9].Vel := 10000;
   PRODUCT_TYPE[3].Motion.Gluing_Rotary_Jig_Axis.Position[1..2].Vel := 20000;
   PRODUCT_TYPE[3].Motion.Gluing_Rotary_Jig_Axis.Position[3..9].Vel := 10000;
   PRODUCT_TYPE[4].Motion.Gluing_Rotary_Jig_Axis.Position[1..2].Vel := 20000;
   PRODUCT_TYPE[4].Motion.Gluing_Rotary_Jig_Axis.Position[3..9].Vel := 10000;
   PRODUCT_TYPE[5].Motion.Gluing_Rotary_Jig_Axis.Position[1..2].Vel := 20000;
   PRODUCT_TYPE[5].Motion.Gluing_Rotary_Jig_Axis.Position[3..9].Vel := 10000;
   PRODUCT_TYPE[6].Motion.Gluing_Rotary_Jig_Axis.Position[1..2].Vel := 20000;
   PRODUCT_TYPE[6].Motion.Gluing_Rotary_Jig_Axis.Position[3..9].Vel := 10000;
   PRODUCT_TYPE[7].Motion.Gluing_Rotary_Jig_Axis.Position[1..2].Vel := 20000;
   PRODUCT_TYPE[7].Motion.Gluing_Rotary_Jig_Axis.Position[3..9].Vel := 10000;
   PRODUCT_TYPE[8].Motion.Gluing_Rotary_Jig_Axis.Position[1..2].Vel := 20000;
   PRODUCT_TYPE[8].Motion.Gluing_Rotary_Jig_Axis.Position[3..9].Vel := 10000;
   PRODUCT_TYPE[9].Motion.Gluing_Rotary_Jig_Axis.Position[1..2].Vel := 20000;
   PRODUCT_TYPE[9].Motion.Gluing_Rotary_Jig_Axis.Position[3..9].Vel := 10000;
   PRODUCT_TYPE[10].Motion.Gluing_Rotary_Jig_Axis.Position[1..2].Vel := 20000;
   PRODUCT_TYPE[10].Motion.Gluing_Rotary_Jig_Axis.Position[3..9].Vel := 10000;
   PRODUCT_TYPE[1].Motion.Ring_Turntable_Axis_2.Position[1].Pos := 3585;
   PRODUCT_TYPE[1].Motion.Ring_Turntable_Axis_2.Position[2].Pos := 48610;
   PRODUCT_TYPE[1].Motion.Ring_Turntable_Axis_2.Position[3].Pos := 93637;
   PRODUCT_TYPE[1].Motion.Ring_Turntable_Axis_2.Position[4].Pos := 138606;
   PRODUCT_TYPE[1].Motion.Ring_Turntable_Axis_2.Position[5].Pos := 183388;
   PRODUCT_TYPE[1].Motion.Ring_Turntable_Axis_2.Position[6].Pos := 228458;
   PRODUCT_TYPE[1].Motion.Ring_Turntable_Axis_2.Position[7].Pos := 273513;
   PRODUCT_TYPE[1].Motion.Ring_Turntable_Axis_2.Position[8].Pos := 318501;
   PRODUCT_TYPE[2].Motion.Ring_Turntable_Axis_2.Position[1].Pos := 3585;
   PRODUCT_TYPE[2].Motion.Ring_Turntable_Axis_2.Position[2].Pos := 48610;
   PRODUCT_TYPE[2].Motion.Ring_Turntable_Axis_2.Position[3].Pos := 93637;
   PRODUCT_TYPE[2].Motion.Ring_Turntable_Axis_2.Position[4].Pos := 138606;
   PRODUCT_TYPE[2].Motion.Ring_Turntable_Axis_2.Position[5].Pos := 183388;
   PRODUCT_TYPE[2].Motion.Ring_Turntable_Axis_2.Position[6].Pos := 228458;
   PRODUCT_TYPE[2].Motion.Ring_Turntable_Axis_2.Position[7].Pos := 273513;
   PRODUCT_TYPE[2].Motion.Ring_Turntable_Axis_2.Position[8].Pos := 318501;
   PRODUCT_TYPE[3].Motion.Ring_Turntable_Axis_2.Position[1].Pos := 3585;
   PRODUCT_TYPE[3].Motion.Ring_Turntable_Axis_2.Position[2].Pos := 48610;
   PRODUCT_TYPE[3].Motion.Ring_Turntable_Axis_2.Position[3].Pos := 93637;
   PRODUCT_TYPE[3].Motion.Ring_Turntable_Axis_2.Position[4].Pos := 138606;
   PRODUCT_TYPE[3].Motion.Ring_Turntable_Axis_2.Position[5].Pos := 183388;
   PRODUCT_TYPE[3].Motion.Ring_Turntable_Axis_2.Position[6].Pos := 228458;
   PRODUCT_TYPE[3].Motion.Ring_Turntable_Axis_2.Position[7].Pos := 273513;
   PRODUCT_TYPE[3].Motion.Ring_Turntable_Axis_2.Position[8].Pos := 318501;
   PRODUCT_TYPE[4].Motion.Ring_Turntable_Axis_2.Position[1].Pos := 3585;
   PRODUCT_TYPE[4].Motion.Ring_Turntable_Axis_2.Position[2].Pos := 48610;
   PRODUCT_TYPE[4].Motion.Ring_Turntable_Axis_2.Position[3].Pos := 93637;
   PRODUCT_TYPE[4].Motion.Ring_Turntable_Axis_2.Position[4].Pos := 138606;
   PRODUCT_TYPE[4].Motion.Ring_Turntable_Axis_2.Position[5].Pos := 183388;
   PRODUCT_TYPE[4].Motion.Ring_Turntable_Axis_2.Position[6].Pos := 228458;
   PRODUCT_TYPE[4].Motion.Ring_Turntable_Axis_2.Position[7].Pos := 273513;
   PRODUCT_TYPE[4].Motion.Ring_Turntable_Axis_2.Position[8].Pos := 318501;
   PRODUCT_TYPE[5].Motion.Ring_Turntable_Axis_2.Position[1].Pos := 3585;
   PRODUCT_TYPE[5].Motion.Ring_Turntable_Axis_2.Position[2].Pos := 48610;
   PRODUCT_TYPE[5].Motion.Ring_Turntable_Axis_2.Position[3].Pos := 93637;
   PRODUCT_TYPE[5].Motion.Ring_Turntable_Axis_2.Position[4].Pos := 138606;
   PRODUCT_TYPE[5].Motion.Ring_Turntable_Axis_2.Position[5].Pos := 183388;
   PRODUCT_TYPE[5].Motion.Ring_Turntable_Axis_2.Position[6].Pos := 228458;
   PRODUCT_TYPE[5].Motion.Ring_Turntable_Axis_2.Position[7].Pos := 273513;
   PRODUCT_TYPE[5].Motion.Ring_Turntable_Axis_2.Position[8].Pos := 318501;
   PRODUCT_TYPE[6].Motion.Ring_Turntable_Axis_2.Position[1].Pos := 3585;
   PRODUCT_TYPE[6].Motion.Ring_Turntable_Axis_2.Position[2].Pos := 48610;
   PRODUCT_TYPE[6].Motion.Ring_Turntable_Axis_2.Position[3].Pos := 93637;
   PRODUCT_TYPE[6].Motion.Ring_Turntable_Axis_2.Position[4].Pos := 138606;
   PRODUCT_TYPE[6].Motion.Ring_Turntable_Axis_2.Position[5].Pos := 183388;
   PRODUCT_TYPE[6].Motion.Ring_Turntable_Axis_2.Position[6].Pos := 228458;
   PRODUCT_TYPE[6].Motion.Ring_Turntable_Axis_2.Position[7].Pos := 273513;
   PRODUCT_TYPE[6].Motion.Ring_Turntable_Axis_2.Position[8].Pos := 318501;
   PRODUCT_TYPE[7].Motion.Ring_Turntable_Axis_2.Position[1].Pos := 3585;
   PRODUCT_TYPE[7].Motion.Ring_Turntable_Axis_2.Position[2].Pos := 48610;
   PRODUCT_TYPE[7].Motion.Ring_Turntable_Axis_2.Position[3].Pos := 93637;
   PRODUCT_TYPE[7].Motion.Ring_Turntable_Axis_2.Position[4].Pos := 138606;
   PRODUCT_TYPE[7].Motion.Ring_Turntable_Axis_2.Position[5].Pos := 183388;
   PRODUCT_TYPE[7].Motion.Ring_Turntable_Axis_2.Position[6].Pos := 228458;
   PRODUCT_TYPE[7].Motion.Ring_Turntable_Axis_2.Position[7].Pos := 273513;
   PRODUCT_TYPE[7].Motion.Ring_Turntable_Axis_2.Position[8].Pos := 318501;
   PRODUCT_TYPE[8].Motion.Ring_Turntable_Axis_2.Position[1].Pos := 3585;
   PRODUCT_TYPE[8].Motion.Ring_Turntable_Axis_2.Position[2].Pos := 48610;
   PRODUCT_TYPE[8].Motion.Ring_Turntable_Axis_2.Position[3].Pos := 93637;
   PRODUCT_TYPE[8].Motion.Ring_Turntable_Axis_2.Position[4].Pos := 138606;
   PRODUCT_TYPE[8].Motion.Ring_Turntable_Axis_2.Position[5].Pos := 183388;
   PRODUCT_TYPE[8].Motion.Ring_Turntable_Axis_2.Position[6].Pos := 228458;
   PRODUCT_TYPE[8].Motion.Ring_Turntable_Axis_2.Position[7].Pos := 273513;
   PRODUCT_TYPE[8].Motion.Ring_Turntable_Axis_2.Position[8].Pos := 318501;
   PRODUCT_TYPE[9].Motion.Ring_Turntable_Axis_2.Position[1].Pos := 3585;
   PRODUCT_TYPE[9].Motion.Ring_Turntable_Axis_2.Position[2].Pos := 48610;
   PRODUCT_TYPE[9].Motion.Ring_Turntable_Axis_2.Position[3].Pos := 93637;
   PRODUCT_TYPE[9].Motion.Ring_Turntable_Axis_2.Position[4].Pos := 138606;
   PRODUCT_TYPE[9].Motion.Ring_Turntable_Axis_2.Position[5].Pos := 183388;
   PRODUCT_TYPE[9].Motion.Ring_Turntable_Axis_2.Position[6].Pos := 228458;
   PRODUCT_TYPE[9].Motion.Ring_Turntable_Axis_2.Position[7].Pos := 273513;
   PRODUCT_TYPE[9].Motion.Ring_Turntable_Axis_2.Position[8].Pos := 318501;
   PRODUCT_TYPE[10].Motion.Ring_Turntable_Axis_2.Position[1].Pos := 3585;
   PRODUCT_TYPE[10].Motion.Ring_Turntable_Axis_2.Position[2].Pos := 48610;
   PRODUCT_TYPE[10].Motion.Ring_Turntable_Axis_2.Position[3].Pos := 93637;
   PRODUCT_TYPE[10].Motion.Ring_Turntable_Axis_2.Position[4].Pos := 138606;
   PRODUCT_TYPE[10].Motion.Ring_Turntable_Axis_2.Position[5].Pos := 183388;
   PRODUCT_TYPE[10].Motion.Ring_Turntable_Axis_2.Position[6].Pos := 228458;
   PRODUCT_TYPE[10].Motion.Ring_Turntable_Axis_2.Position[7].Pos := 273513;
   PRODUCT_TYPE[10].Motion.Ring_Turntable_Axis_2.Position[8].Pos := 318501;
   PRODUCT_TYPE[1].Motion.Ring_Turntable_Axis_2.Position[1..8].Vel := 10000;
   PRODUCT_TYPE[2].Motion.Ring_Turntable_Axis_2.Position[1..8].Vel := 10000;
   PRODUCT_TYPE[3].Motion.Ring_Turntable_Axis_2.Position[1..8].Vel := 10000;
   PRODUCT_TYPE[4].Motion.Ring_Turntable_Axis_2.Position[1..8].Vel := 10000;
   PRODUCT_TYPE[5].Motion.Ring_Turntable_Axis_2.Position[1..8].Vel := 10000;
   PRODUCT_TYPE[6].Motion.Ring_Turntable_Axis_2.Position[1..8].Vel := 10000;
   PRODUCT_TYPE[7].Motion.Ring_Turntable_Axis_2.Position[1..8].Vel := 10000;
   PRODUCT_TYPE[8].Motion.Ring_Turntable_Axis_2.Position[1..8].Vel := 10000;
   PRODUCT_TYPE[9].Motion.Ring_Turntable_Axis_2.Position[1..8].Vel := 10000;
   PRODUCT_TYPE[10].Motion.Ring_Turntable_Axis_2.Position[1..8].Vel := 10000;
END_DATA_BLOCK
